(*Nocken speichern und Rest ignorieren*)
IF	fb_ton_end.Q AND
	(MEMCMP(ADR(gst_datensatz_copy.st_wkz.nockenschaltwerk_bestueckachse), ADR(gst_datensatz.st_wkz.nockenschaltwerk_bestueckachse), SIZEOF(gst_datensatz_copy.st_wkz.nockenschaltwerk_bestueckachse)) <> 0 ) THEN
	FOR j := 0 TO MAX_NOCKENGERUEST DO	(*nur die Nocken begin und end speichern*)
		IF	gst_datensatz_copy.st_wkz.nockenschaltwerk_bestueckachse.arr_nocken[j].r_cam_begin<>gst_datensatz.st_wkz.nockenschaltwerk_bestueckachse.arr_nocken[j].r_cam_begin OR
			gst_datensatz_copy.st_wkz.nockenschaltwerk_bestueckachse.arr_nocken[j].r_cam_end<>gst_datensatz.st_wkz.nockenschaltwerk_bestueckachse.arr_nocken[j].r_cam_end THEN
			i16_auftrag:=SCHREIBE_WKZ;
		END_IF
	END_FOR
	gst_datensatz_copy.st_wkz.nockenschaltwerk_bestueckachse:=gst_datensatz.st_wkz.nockenschaltwerk_bestueckachse;
END_IF

(*Wkz Daten speichern*)
IF	fb_ton_end.Q AND
	gi16_maschinenstatusinfo <> STATUS_MASCHINE_ARBEITET AND
	(MEMCMP(ADR(gst_datensatz_copy.st_wkz), ADR(gst_datensatz.st_wkz), SIZEOF(gst_datensatz_copy.st_wkz)) <> 0 ) THEN
	i16_auftrag:=SCHREIBE_WKZ;
END_IF

(*Band Daten speichern*)
IF	fb_ton_end.Q AND
	gi16_maschinenstatusinfo <> STATUS_MASCHINE_ARBEITET AND
	(MEMCMP(ADR(gst_datensatz_copy.st_band), ADR(gst_datensatz.st_band), SIZEOF(gst_datensatz_copy.st_band)) <> 0 ) THEN
	i16_auftrag:=SCHREIBE_BAND;
END_IF

(*Wt Daten speichern*)
IF	fb_ton_end.Q AND
	gi16_maschinenstatusinfo <> STATUS_MASCHINE_ARBEITET AND
	(MEMCMP(ADR(gst_datensatz_copy.st_wt), ADR(gst_datensatz.st_wt), SIZEOF(gst_datensatz_copy.st_wt)) <> 0 ) THEN
	i16_auftrag:=SCHREIBE_WT;
END_IF

(*Maschinen Daten speichern*)
IF	fb_ton_end.Q AND
	gi16_maschinenstatusinfo <> STATUS_MASCHINE_ARBEITET AND
	(MEMCMP(ADR(gst_datensatz_copy.st_md), ADR(gst_datensatz.st_md), SIZEOF(gst_datensatz_copy.st_md)) <> 0 ) THEN
	i16_auftrag:=SCHREIBE_MD;
	hm_md_speichern:=FALSE;
END_IF
END_ACTION
ACTION generiere_bestueckbild:
(* Step 1: erzeuge eine Liste mit allen unseren Pins *)
st_akt_bestueckprogramm.i32_anzahl := 0;

FOR i := 0 TO gst_bestueckbild.i32_anzahl_pins - 1 BY 1
DO
	IF (gst_bestueckbild.st_pins[i].typ = gst_datensatz.st_md.s_aktuelles_band) THEN
		st_akt_bestueckprogramm.lr_y[st_akt_bestueckprogramm.i32_anzahl] := gst_bestueckbild.st_pins[i].lr_y;
		st_akt_bestueckprogramm.lr_z[st_akt_bestueckprogramm.i32_anzahl] := gst_bestueckbild.st_pins[i].lr_z;
		st_akt_bestueckprogramm.i16_b[st_akt_bestueckprogramm.i32_anzahl] := 1;

		st_akt_bestueckprogramm.i32_anzahl  := st_akt_bestueckprogramm.i32_anzahl + 1;
	END_IF
END_FOR


(* Step 2: Sortieren: Bubblesort by Z *)
sort_akt();

(* Einragen in die globale Sruktur *)
gst_datensatz.st_bestueckprogramm := st_akt_bestueckprogramm;
gst_datensatz.st_md.s_aktueller_isk := gst_bestueckbild.s_isknummer;
END_ACTION
ACTION Hub_Faktor_ermitteln:
 (*ermitteln der maximal zu bestückenden Pins eines Bestückbildes=========================*)

FOR n := 0 TO 14 DO
	s_HelpBand[n]:='';
	i32_Anzahl[n]:=0;
END_FOR
i32_maxAnzahl := 0;

FOR n := 0 TO 14 DO
	FOR m := 0 TO gst_bestueckbild.i32_anzahl_pins - 1 DO
		IF	gst_bestueckbild.st_pins[m].typ <> s_HelpBand[0] AND
			gst_bestueckbild.st_pins[m].typ <> s_HelpBand[1] AND
			gst_bestueckbild.st_pins[m].typ <> s_HelpBand[2] AND
			gst_bestueckbild.st_pins[m].typ <> s_HelpBand[3] AND
			gst_bestueckbild.st_pins[m].typ <> s_HelpBand[4] AND
			gst_bestueckbild.st_pins[m].typ <> s_HelpBand[5] AND
			gst_bestueckbild.st_pins[m].typ <> s_HelpBand[6] AND
			gst_bestueckbild.st_pins[m].typ <> s_HelpBand[7] AND
			gst_bestueckbild.st_pins[m].typ <> s_HelpBand[8] AND
			gst_bestueckbild.st_pins[m].typ <> s_HelpBand[9] AND
			gst_bestueckbild.st_pins[m].typ <> s_HelpBand[10] AND
			gst_bestueckbild.st_pins[m].typ <> s_HelpBand[11] AND
			gst_bestueckbild.st_pins[m].typ <> s_HelpBand[12] AND
			gst_bestueckbild.st_pins[m].typ <> s_HelpBand[13] AND
			gst_bestueckbild.st_pins[m].typ <> s_HelpBand[14] THEN
			s_HelpBand[n]:=gst_bestueckbild.st_pins[m].typ;
		END_IF
	END_FOR
END_FOR

FOR n := 0 TO 14 DO
	FOR m := 0 TO gst_bestueckbild.i32_anzahl_pins - 1 DO
		IF gst_bestueckbild.st_pins[m].typ = s_HelpBand[n] AND s_HelpBand[n] <>'' THEN
			i32_Anzahl[n]:=i32_Anzahl[n]+1;
		END_IF
	END_FOR
	IF	i32_Anzahl[n]>i32_maxAnzahl THEN
		i32_maxAnzahl:=i32_Anzahl[n];
	END_IF
END_FOR

(* Faktor für die Hubzahl*)
lr_min_FaktorHub:=100/gst_datensatz.st_wkz.r_auto;

IF	i32_maxAnzahl > 0  THEN

	lr_FaktorHub:=(DINT_TO_LREAL(st_akt_bestueckprogramm.i32_anzahl) / DINT_TO_LREAL(i32_maxAnzahl)) * 1.2;
	IF	lr_FaktorHub > 1 THEN
		lr_FaktorHub:=1;
	END_IF
	IF	lr_FaktorHub < lr_min_FaktorHub THEN 	(*Bestückgeschwindigkeit nur um maximal 100Hub verringern*)
		lr_FaktorHub:=lr_min_FaktorHub;
	END_IF
ELSE
	lr_FaktorHub:=1;
END_IF
END_ACTION
ACTION Hub_Faktor_ermitteln_halbauto:
 (*ermitteln der maximal zu bestückenden Pins eines Bestückbildes=========================*)
n:=-1;
i32_maxAnzahl := 0;
FOR n := 0 TO 14 DO
	i32_Anzahl[n]:=gst_bestueckbild_halbauto.Wkz[n].i32_anzahl;
	IF	i32_Anzahl[n]>i32_maxAnzahl THEN
		i32_maxAnzahl:=i32_Anzahl[n];
	END_IF
END_FOR

(* Faktor für die Hubzahl*)
lr_min_FaktorHub:=100/gst_datensatz.st_wkz.r_auto;

IF	i32_maxAnzahl > 0  THEN

	lr_FaktorHub:=(DINT_TO_LREAL(gst_datensatz.st_bestueckprogramm.i32_anzahl) / DINT_TO_LREAL(i32_maxAnzahl)) * 1.35;
	IF	lr_FaktorHub > 1 THEN
		lr_FaktorHub:=1;
	END_IF
	IF	lr_FaktorHub < lr_min_FaktorHub THEN 	(*Bestückgeschwindigkeit nur um maximal 100Hub verringern*)
		lr_FaktorHub:=lr_min_FaktorHub;
	END_IF
ELSE
	lr_FaktorHub:=1;
END_IF
END_ACTION
ACTION path:
IF	s_Projekt_path <> '' THEN
	IF	FIND(s_md_path,':') = 0 THEN
		s_md_path 	:= CONCAT(s_Projekt_path,s_md_path);
	END_IF
	IF	FIND(s_tools_path,':') = 0 THEN
		s_tools_path 	:= CONCAT(s_Projekt_path,s_tools_path);
	END_IF
END_IF
END_ACTION
ACTION sort_akt:
FOR i := st_akt_bestueckprogramm.i32_anzahl -1 TO 1  BY -1
DO
	FOR k := 0 TO i -1 BY 1
	DO
		CASE gst_bestueckbild.enu_richtung OF

			(* Y Spalte Minus nach Plus: Bei gleichem Y: Z minus nach Plus *)
			YMinus_nach_YPlus_ZMinus_nach_ZPlus:
				IF F_Vergleich_LReal(st_akt_bestueckprogramm.lr_y[k+1] , st_akt_bestueckprogramm.lr_y[k]) THEN
					b_sort_swap := st_akt_bestueckprogramm.lr_z[k+1] < st_akt_bestueckprogramm.lr_z[k];
				ELSE
					b_sort_swap := st_akt_bestueckprogramm.lr_y[k+1] < st_akt_bestueckprogramm.lr_y[k];
				END_IF

			(* Y Spalte Minus nach Plus: Bei gleichem Y: Z Plus nach Minus *)
			YMinus_nach_YPlus_ZPlus_nach_ZMinus:
				IF F_Vergleich_LReal(st_akt_bestueckprogramm.lr_y[k+1] , st_akt_bestueckprogramm.lr_y[k]) THEN
					b_sort_swap := st_akt_bestueckprogramm.lr_z[k+1] > st_akt_bestueckprogramm.lr_z[k];
				ELSE
					b_sort_swap := st_akt_bestueckprogramm.lr_y[k+1]< st_akt_bestueckprogramm.lr_y[k];
				END_IF

			(* Y Spalte Plus nach Minus: Bei gleichem Y: Z Minus nach Plus *)
			YPlus_nach_YMinus_ZMinus_nach_ZPlus:
				IF F_Vergleich_LReal(st_akt_bestueckprogramm.lr_y[k+1] , st_akt_bestueckprogramm.lr_y[k]) THEN
					b_sort_swap := st_akt_bestueckprogramm.lr_z[k+1] < st_akt_bestueckprogramm.lr_z[k];
				ELSE
					b_sort_swap := st_akt_bestueckprogramm.lr_y[k+1] > st_akt_bestueckprogramm.lr_y[k];
				END_IF

			(* Y Spalte Plus nach Minus: Bei gleichem Y: Z Plus nach Minus *)
			YPlus_nach_YMinus_ZPlus_nach_ZMinus:
				IF F_Vergleich_LReal(st_akt_bestueckprogramm.lr_y[k+1] , st_akt_bestueckprogramm.lr_y[k]) THEN
					b_sort_swap := st_akt_bestueckprogramm.lr_z[k+1] > st_akt_bestueckprogramm.lr_z[k];
				ELSE
					b_sort_swap := st_akt_bestueckprogramm.lr_y[k+1] > st_akt_bestueckprogramm.lr_y[k];
				END_IF
		END_CASE

		IF b_sort_swap THEN
			(* Tauschen k + 1 <--> k *)
			swap_a := k; swap_b := k+1;	swap_in_akt();
		END_IF

	END_FOR
END_FOR
END_ACTION
ACTION subr_Wkz_Band_Wt_schreiben:
(* ======================================Schrittkette======================================== *)
fb_state_entry2(	i16_pos:= 1 );

CASE fb_state_entry2.i16_step OF
(*=======================================================*)
	0:

		fb_wkz_band_wt_schreiben.Start := FALSE;

		(*-----------------------Weiterschaltbedingungen----------------------------*)
		fb_state_entry2.i16_next_step := BEREIT;

(*=======================================================*)
	BEREIT:	(* Warte auf Änderung *)

		(*-----------------------Weiterschaltbedingungen----------------------------*)
		IF gst_datensatz.st_md.s_aktuelles_wkz <> s_name_alt_wkz OR
		    gst_datensatz.st_md.s_aktuelles_band <> s_name_alt_band OR
		    gst_datensatz.st_md.s_aktueller_wt <> s_name_alt_wt THEN
			s_name_alt_wkz := gst_datensatz.st_md.s_aktuelles_wkz;
			s_name_alt_band :=gst_datensatz.st_md.s_aktuelles_band;
			s_name_alt_wt := gst_datensatz.st_md.s_aktueller_wt;
			fb_state_entry2.i16_next_step := 200;
		END_IF

(*=======================================================*)
	200: (* Aktuelles WKZ in txt Datei schreiben *)
		IF fb_state_entry2.E THEN
			fb_wkz_band_wt_schreiben.ExportStr := gst_datensatz.st_md.s_aktuelles_wkz;
			fb_wkz_band_wt_schreiben.FileName := 'Aktuelles_Wkz.txt';
			fb_wkz_band_wt_schreiben.Start := TRUE;
		END_IF

		(*-----------------------Weiterschaltbedingungen----------------------------*)
		IF fb_wkz_band_wt_schreiben.Busy THEN
			fb_wkz_band_wt_schreiben.Start := FALSE;
			fb_state_entry2.i16_next_step := 210;
		END_IF

(*=======================================================*)
	210: (* warte auf fertig *)

		(*-----------------------Weiterschaltbedingungen----------------------------*)
		IF fb_wkz_band_wt_schreiben.Done THEN
			fb_state_entry2.i16_next_step := 300;
		END_IF

(*=======================================================*)
	300: (* Aktuelles WKZ in txt Datei schreiben *)
		IF fb_state_entry2.E THEN
			fb_wkz_band_wt_schreiben.ExportStr := gst_datensatz.st_md.s_aktuelles_band;
			fb_wkz_band_wt_schreiben.FileName := 'Aktuelles_Band.txt';
			fb_wkz_band_wt_schreiben.Start := TRUE;
		END_IF

		(*-----------------------Weiterschaltbedingungen----------------------------*)
		IF fb_wkz_band_wt_schreiben.Busy THEN
			fb_wkz_band_wt_schreiben.Start := FALSE;
			fb_state_entry2.i16_next_step := 310;
		END_IF

(*=======================================================*)
	310: (* warte auf fertig *)

		(*-----------------------Weiterschaltbedingungen----------------------------*)
		IF fb_wkz_band_wt_schreiben.Done THEN
			fb_state_entry2.i16_next_step := 400;
		END_IF

(*=======================================================*)
	400: (* Aktuellen Wt in txt Datei schreiben *)
		IF fb_state_entry2.E THEN
			fb_wkz_band_wt_schreiben.ExportStr := gst_datensatz.st_md.s_aktueller_wt;
			fb_wkz_band_wt_schreiben.FileName := 'Aktueller_Wt.txt';
			fb_wkz_band_wt_schreiben.Start := TRUE;
		END_IF

		(*-----------------------Weiterschaltbedingungen----------------------------*)
		IF fb_wkz_band_wt_schreiben.Busy THEN
			fb_wkz_band_wt_schreiben.Start := FALSE;
			fb_state_entry2.i16_next_step := 410;
		END_IF

(*=======================================================*)
	410: (* warte auf fertig *)

		(*-----------------------Weiterschaltbedingungen----------------------------*)
		IF fb_wkz_band_wt_schreiben.Done THEN
			fb_state_entry2.i16_next_step := BEREIT;
		END_IF

END_CASE

fb_state_entry2(i16_pos:= 2 );

fb_wkz_band_wt_schreiben(
	Start:= ,
	ExportStr:= ,
	FileName:= ,
	Path:= 'D:\BBgen\',
	Mode:= 2,
	Ready=> , 
	Busy=> , 
	Done=> ,
	Error=> );
END_ACTION
ACTION swap_in_akt:
lr_tmp := st_akt_bestueckprogramm.lr_y[swap_a];
st_akt_bestueckprogramm.lr_y[swap_a] := st_akt_bestueckprogramm.lr_y[swap_b];
st_akt_bestueckprogramm.lr_y[swap_b] := lr_tmp;

lr_tmp := st_akt_bestueckprogramm.lr_z[swap_a];
st_akt_bestueckprogramm.lr_z[swap_a] := st_akt_bestueckprogramm.lr_z[swap_b];
st_akt_bestueckprogramm.lr_z[swap_b] := lr_tmp;

i16_tmp := st_akt_bestueckprogramm.i16_b[swap_a];
st_akt_bestueckprogramm.i16_b[swap_a] := st_akt_bestueckprogramm.i16_b[swap_b];
st_akt_bestueckprogramm.i16_b[swap_b] := i16_tmp;
END_ACTION
ACTION wkz_gruppe_kompatibel:
(*Gruppe löschen wenn ein neues Werkzeug ausgewählt wird*)
IF	gst_datensatz_copy.st_md.s_aktuelles_wkz<>gst_datensatz.st_md.s_aktuelles_wkz THEN
	i:=-1;
	FOR i := 0 TO 4 DO
		gst_datensatz.st_md.st_wkz_gruppe[i].s_wkz := '';
		gst_datensatz.st_md.st_wkz_gruppe[i].i16_wkz_gruppe_kompatibel := 0;
		gst_datensatz.st_md.st_wkz_gruppe[i].s_Band := '';
		gst_datensatz.st_md.st_wkz_gruppe[i].i32_Wkz_nr := -1;
		gst_datensatz.st_md.st_wkz_gruppe[i].i32_Anzahl := -1;
	END_FOR
END_IF

(*Fehler*)
IF	state =0 THEN
	k:=-1;
	sm_Wkz_Gruppe_nicht_zugeordnet:=FALSE;
	sm_Wkz_nicht_kompatibel:=FALSE;
	FOR k := 0 TO 4 DO
		i:=-1;
		FOR i := 0 TO 4 DO
			IF	gst_datensatz.st_md.st_wkz_gruppe[k].s_wkz <> '' AND
				gst_datensatz.st_md.st_wkz_gruppe[i].s_wkz <> '' AND
				gst_datensatz.st_md.st_wkz_gruppe[k].i16_wkz_gruppe_kompatibel <>gst_datensatz.st_md.st_wkz_gruppe[i].i16_wkz_gruppe_kompatibel THEN
				sm_Wkz_nicht_kompatibel:=TRUE;
			END_IF
		END_FOR

		IF	gst_datensatz.st_md.st_wkz_gruppe[k].s_wkz <> '' AND
			gst_datensatz.st_md.st_wkz_gruppe[k].i16_wkz_gruppe_kompatibel = 0 THEN
			sm_Wkz_Gruppe_nicht_zugeordnet:=TRUE;
		END_IF

	END_FOR
END_IF

(*==========================================================================================*)
b_Wkz_Gruppe_gebildet:=
	NOT sm_Wkz_nicht_kompatibel AND
	gst_datensatz.st_md.st_wkz_gruppe[0].s_wkz <> '' AND
	gst_datensatz.st_md.st_wkz_gruppe[1].s_wkz <> '';

i16_anzahl_Wkz_Gruppen:=0;
k:=-1;
FOR k := 0 TO 4 DO
	IF	gst_datensatz.st_md.st_wkz_gruppe[k].s_wkz <> ''	THEN
		i16_anzahl_Wkz_Gruppen:=i16_anzahl_Wkz_Gruppen + 1;
	END_IF
END_FOR

(*==========================================================================================*)
CASE state OF
0:	(* Auslesen wenn ein neues Wkz ausgewählt wird*)
	fb_xml_srv_read.bExecute:= FALSE;
	k:=-1;
	FOR k := 0 TO 4 DO
		IF	state =0 AND
			st_wkz_gruppe_copy[k].s_wkz<>gst_datensatz.st_md.st_wkz_gruppe[k].s_wkz THEN

			IF	gst_datensatz.st_md.st_wkz_gruppe[k].s_wkz='' THEN
				st_wkz_gruppe_copy[k].s_wkz:=gst_datensatz.st_md.st_wkz_gruppe[k].s_wkz;
			ELSE
				i32_neues_Wkz:=k;
				state:=10;
			END_IF

			gst_datensatz.st_md.st_wkz_gruppe[k].i16_wkz_gruppe_kompatibel:=0;
			st_wkz_gruppe_copy[k].i16_wkz_gruppe_kompatibel:=0;
			gst_datensatz.st_md.st_wkz_gruppe[k].s_Band := '';
			gst_datensatz.st_md.st_wkz_gruppe[k].i32_Wkz_nr := -1;
			gst_datensatz.st_md.st_wkz_gruppe[k].i32_Anzahl := -1;

		END_IF
	END_FOR

10:	(*Start auslesen*)
	nErrId := 0;
	fb_xml_srv_read.sFilePath:= 'D:\BBgen\Wkz\';
	fb_xml_srv_read.sFilePath:= CONCAT(fb_xml_srv_read.sFilePath,gst_datensatz.st_md.st_wkz_gruppe[i32_neues_Wkz].s_wkz);
	fb_xml_srv_read.sFilePath:= CONCAT(fb_xml_srv_read.sFilePath,'.xml');
	fb_xml_srv_read.sXPath := '/root/gst_datensatz.st_wkz/I16_WKZ_GRUPPE_KOMPATIBEL';
	fb_xml_srv_read.sSymName:= '.gst_datensatz.st_md.st_wkz_gruppe[';
	fb_xml_srv_read.sSymName:= CONCAT(fb_xml_srv_read.sSymName,DINT_TO_STRING(i32_neues_Wkz));
	fb_xml_srv_read.sSymName:= CONCAT(fb_xml_srv_read.sSymName,'].i16_wkz_gruppe_kompatibel');
	fb_xml_srv_read.bExecute:= TRUE;

	IF fb_xml_srv_read.bBusy THEN
		fb_xml_srv_read.bExecute:= FALSE;
		state := 20;
	END_IF

20:	(* Lesevorgang erfolgreich? *)
	IF NOT fb_xml_srv_read.bBusy THEN
		IF NOT fb_xml_srv_read.bError THEN
			state := 0;
			st_wkz_gruppe_copy[i32_neues_Wkz].s_wkz:=gst_datensatz.st_md.st_wkz_gruppe[i32_neues_Wkz].s_wkz;
			st_wkz_gruppe_copy[i32_neues_Wkz].i16_wkz_gruppe_kompatibel:=gst_datensatz.st_md.st_wkz_gruppe[i32_neues_Wkz].i16_wkz_gruppe_kompatibel;
		ELSE	(* Fehler *)
			nErrId := fb_xml_srv_read.nErrId;
			state := FEHLER;
		END_IF
	END_IF

FEHLER:
	state := 0;
	st_wkz_gruppe_copy[i32_neues_Wkz].s_wkz:=gst_datensatz.st_md.st_wkz_gruppe[i32_neues_Wkz].s_wkz;
END_CASE
END_ACTION

(* POU EPT Lib/Funktionsbausteine/ST_StateEntry, ST *)
FUNCTION_BLOCK ST_StateEntry
VAR
	arr_last_step_history	: ARRAY[0..31] OF STRING(110);
	i 					: INT := 0;
	last_pos 				: INT := 0;
	interner_step			: INT := 0;
	s_stepTime 			: STRING;
END_VAR
VAR_OUTPUT
	i16_last_step 			: enum_step_nr := INIT_OBJ;	(* Der Schritt vor diesem Schritt *)
	i16_step 				: enum_step_nr := INIT_OBJ;	(* Diese variable soll vom "case step of" verwendet werden *)
	E					: BOOL;					(* Aktiv bei betreten des Steps *)
	X					: BOOL;					(* Aktiv beim verlassen des Steps *)
	b_error 				: BOOL := FALSE;			(* Ablauf Pos 1,2,1,2,1,2,... nicht richtig *)
	fb_ton_Step			: TON;
END_VAR
VAR_INPUT
	i16_next_step 		: enum_step_nr := INIT_OBJ;	(* Nächster schritt *)
	i16_pos 				: INT;					(* Pos = 1: Aufruf vor dem Case step of ---  Pos = 2: Aufruf nach dem Case step of*)
	s_debugtext			: STRING(100);
END_VAR
VAR CONSTANT
	t_MaxStepTime		: TIME := T#60S;
END_VAR
(*stepTime ermitteln*)
fb_ton_Step(IN:= , PT:=t_MaxStepTime , Q=>  , ET=> );
IF	i16_step = i16_next_step THEN
	fb_ton_Step.IN:=TRUE;
END_IF

IF NOT b_error THEN
	CASE interner_step OF
		0:
			(* Mitten im Schritt drin *)
			X := FALSE;
			E := FALSE;


			(* Schritt wird verlassen *)
			IF i16_step <> i16_next_step AND i16_pos = 1 THEN
				subrDebugtext();
				interner_step := 10;
				X := TRUE;
				E := FALSE;
				fb_ton_Step.IN:=FALSE;
			END_IF

		10:
			(* Eintritt in neuen Schritt *)
			IF i16_pos = 1 THEN
				X := FALSE;
				E := TRUE;

				(* Schalte Schritt weiter *)
				i16_last_step := i16_step;
				i16_step := i16_next_step;
				(* Baue Statehistory *)

				IF  E THEN
					FOR i:= 31 TO 1 BY -1 DO
						arr_last_step_history[i] := arr_last_step_history[i-1];
					END_FOR
					arr_last_step_history[0] := '';
					s_stepTime:='';
					s_debugtext:='';
				END_IF

				interner_step := 0;

			END_IF
	END_CASE
END_IF

IF 	(fb_ton_Step.ET >= T#200ms AND arr_last_step_history[0] = '') OR	(* Am Anfang Debugtext schreiben, damit etwas drin steht *)
	(fb_ton_Step.Q AND s_stepTime <> '>1m') THEN	(* Debugtext schreiben, wenn t_MaxStepTime erreicht wird *)
	subrDebugtext();
END_IF

(* Prüfe Baustein *)
IF 	i16_pos = last_pos THEN
	b_error := TRUE;
END_IF

last_pos := i16_pos;
END_FUNCTION_BLOCK
ACTION subrDebugtext:
s_stepTime:=ET_TO_STRING(fb_ton_Step.ET);
IF 	fb_ton_Step.ET >= t_MaxStepTime THEN
	s_stepTime:=CONCAT('>',s_StepTime);
END_IF

(* history zusammenbauen aus StepNr, StepTime und debugtext*)
CASE i16_step OF
	INIT_OBJ :			arr_last_step_history[0]:='INIT_OBJ';
	INIT :				arr_last_step_history[0]:='INIT';
	BEREIT :				arr_last_step_history[0]:='BEREIT';
	FEHLER :			arr_last_step_history[0]:='FEHLER';
	STOP :				arr_last_step_history[0]:='STOP';
	STILLSTAND :		arr_last_step_history[0]:='STILLSTAND';
	HALT :				arr_last_step_history[0]:='HALT';
	HANDRAD :			arr_last_step_history[0]:='HANDRAD';
	MOTORBREMSE_AUF :	arr_last_step_history[0]:='MOTORBREMSE_AUF';
	MOTORBREMSE_ZU :	arr_last_step_history[0]:='MOTORBREMSE_ZU';
	LUEFTEN :			arr_last_step_history[0]:='LUEFTEN';
	REGELN :			arr_last_step_history[0]:='REGELN';
	INBETRIEBNAHME :		arr_last_step_history[0]:='INBETRIEBNAHME';
	(* Zylinder *)
	ZYL_INIT :			arr_last_step_history[0]:='ZYL_INIT';
	GESTOPPT :			arr_last_step_history[0]:='GESTOPPT';
	EINGEFAHREN :		arr_last_step_history[0]:='EINGEFAHREN';
	BEWEGUNG_AUSFAHREN :		arr_last_step_history[0]:='BEWEGUNG_AUSFAHREN';
	AUSGEFAHREN :		arr_last_step_history[0]:='AUSGEFAHREN';
	BEWEGUNG_EINFAHREN :		arr_last_step_history[0]:='BEWEGUNG_EINFAHREN';
	MITTEGEFAHREN :		arr_last_step_history[0]:='MITTEGEFAHREN';
	BEWEGUNG_MITTE  :	arr_last_step_history[0]:='BEWEGUNG_MITTE';
	LUFTLOS :			arr_last_step_history[0]:='LUFTLOS';
	ZYL_FEHLER :		arr_last_step_history[0]:='ZYL_FEHLER';
	DIREKT_EINFAHREN :	arr_last_step_history[0]:='DIREKT_EINFAHREN';
	DIREKT_AUSFAHREN :	arr_last_step_history[0]:='DIREKT_AUSFAHREN';
ELSE
	arr_last_step_history[0] := INT_TO_STRING(i16_step);
END_CASE

IF 	s_stepTime ='0ms' OR s_stepTime =''THEN
	s_stepTime:='3ms';		(*damit nicht 0 drin steht*)
END_IF
arr_last_step_history[0] := CONCAT(arr_last_step_history[0],':  ');
arr_last_step_history[0] := CONCAT(arr_last_step_history[0],s_stepTime);
arr_last_step_history[0] := CONCAT(arr_last_step_history[0],': ');
arr_last_step_history[0] := CONCAT(arr_last_step_history[0],s_debugtext);
END_ACTION

(* POU EPT Lib/Funktionen/ET_TO_STRING, ST *)
FUNCTION ET_TO_STRING :STRING
VAR_INPUT
	et		:TIME;
END_VAR

VAR
	i16_LEN	:INT;
END_VAR
ET_TO_STRING:=TIME_TO_STRING(et);
ET_TO_STRING:=DELETE(ET_TO_STRING,2,1);

IF 	et> t#60s THEN
	ET_TO_STRING:=LEFT(ET_TO_STRING,FIND(ET_TO_STRING,'s'));
END_IF
END_FUNCTION

(* POU Gemeinsamkeiten17xx/BBGen/ST_BBGenXMLFile, ST *)
FUNCTION_BLOCK ST_BBGenXMLFile
VAR_INPUT
	bQuit								: BOOL;
	(* ISK *)
	start_lesen_isk						: BOOL;
	start_schreiben_isk					: BOOL;

	(* Wkz *)
	start_lesen_wkz						: BOOL;
	start_schreiben_wkz					: BOOL;

	(* Bestueckbild wird nur gelesen *)
	start_lesen_bestueckbild				: BOOL;
	start_schreiben_bestueckbild			: BOOL;

	(* Bestueckbild Halbautomatik wird nur gelesen *)
	start_lesen_bestueckbild_halbauto				: BOOL;
	start_schreiben_bestueckbild_halbauto			: BOOL;

	(* Maschinendaten *)
	start_lesen_md						: BOOL;
	start_schreiben_md					: BOOL;
	start_schreiben_md_backup			: BOOL;

	(* Banddaten *)
	start_lesen_band						: BOOL;
	start_schreiben_band					: BOOL;

	(* Wt-Daten *)
	start_lesen_wt						: BOOL;
	start_schreiben_wt						: BOOL;

	(* Wo liegen die Dateien *)
	s_path								: STRING(255);

	(* Welche Dateien? *)
	s_bestueckbild						: STRING(50);
	s_wkz								: STRING(50);
	s_isk								: STRING(50);
	s_md								: STRING(50);
	s_md_backup						: STRING(50);
	s_band								: STRING(50);
	s_wt									: STRING(50);
END_VAR
VAR_OUTPUT
	fertig_lesen							: BOOL;
	fertig_schreiben						: BOOL;

	bError								: BOOL;
	nErrId								: UDINT;
END_VAR
VAR
	fb_state_entry							: ST_StateEntry;
	fb_ton_quitt							: TON;
	fb_xml_srv_write						: FB_XmlSrvWriteByName;
	fb_xml_srv_read						: FB_XmlSrvReadByName;
	s_file								: STRING(255);

END_VAR
fb_ton_quitt(IN:= , PT:= t#50ms, Q=> , ET=> );

(* ======================================Schrittkette======================================== *)
fb_state_entry(
	i16_next_step:= ,
	i16_pos:= 1,
	s_debugtext:= ,
	E=> ,
	X=> ,
	i16_step=> ,
	i16_last_step=> );


CASE fb_state_entry.i16_step OF
(*=======================================================*)
	0:
		bError := FALSE;
		nErrId := 0;

		fertig_lesen := FALSE;
		fertig_schreiben := FALSE;

		fb_state_entry.i16_next_step := 10;

(*=======================================================*)
	10:	(* Auslesen der Daten aus den XML-Files *)
		(* Daten lesen *)
		IF start_lesen_isk THEN
			s_file := CONCAT(s_path, s_isk);
			s_file := CONCAT(s_file,'.xml');
			fb_xml_srv_read.sSymName := '.gst_datensatz.st_isk';
			fb_xml_srv_read.sXPath := '/root/gst_datensatz.st_isk';
			fb_state_entry.i16_next_step := 100;
		ELSIF start_lesen_bestueckbild THEN
			s_file := CONCAT(s_path, s_bestueckbild);
			s_file := CONCAT(s_file,'.xml');
			fb_xml_srv_read.sSymName := '.gst_bestueckbild';
			fb_xml_srv_read.sXPath := '/root/gst_bestueckbild';
			fb_state_entry.i16_next_step := 100;

		ELSIF start_lesen_bestueckbild_halbauto THEN
			s_file := CONCAT(s_path, s_bestueckbild);
			s_file := CONCAT(s_file,'.xml');
			fb_xml_srv_read.sSymName := '.gst_bestueckbild_halbauto';
			fb_xml_srv_read.sXPath := '/root/gst_bestueckbild_halbauto';
			fb_state_entry.i16_next_step := 100;

		ELSIF start_lesen_wkz THEN
			s_file := CONCAT(s_path, s_wkz);
			s_file := CONCAT(s_file,'.xml');
			fb_xml_srv_read.sSymName := '.gst_datensatz.st_wkz';
			fb_xml_srv_read.sXPath := '/root/gst_datensatz.st_wkz';
			fb_state_entry.i16_next_step := 100;
		ELSIF start_lesen_md THEN
			s_file := CONCAT(s_path, s_md);
			s_file := CONCAT(s_file,'.xml');
			fb_xml_srv_read.sSymName := '.gst_datensatz.st_md';
			fb_xml_srv_read.sXPath := '/root/gst_datensatz.st_md';
			fb_state_entry.i16_next_step := 100;
		ELSIF start_lesen_band THEN
			s_file := CONCAT(s_path, s_band);
			s_file := CONCAT(s_file,'.xml');
			fb_xml_srv_read.sSymName := '.gst_datensatz.st_band';
			fb_xml_srv_read.sXPath := '/root/gst_datensatz.st_band';
			fb_state_entry.i16_next_step := 100;
		ELSIF start_lesen_wt THEN
			s_file := CONCAT(s_path, s_wt);
			s_file := CONCAT(s_file,'.xml');
			fb_xml_srv_read.sSymName := '.gst_datensatz.st_wt';
			fb_xml_srv_read.sXPath := '/root/gst_datensatz.st_wt';
			fb_state_entry.i16_next_step := 100;
		END_IF

		(* Daten schreiben *)
		IF start_schreiben_isk THEN
			s_file := CONCAT(s_path, s_isk);
			s_file := CONCAT(s_file,'.xml');
			fb_xml_srv_write.sSymName := '.gst_datensatz.st_isk';
			fb_xml_srv_write.sXPath := '/root/gst_datensatz.st_isk';
			fb_state_entry.i16_next_step := 200;
		ELSIF start_schreiben_bestueckbild THEN
			s_file := CONCAT(s_path, s_bestueckbild);
			s_file := CONCAT(s_file,'.xml');
			fb_xml_srv_write.sSymName := '.gst_bestueckbild';
			fb_xml_srv_write.sXPath := '/root/gst_bestueckbild';
			fb_state_entry.i16_next_step := 200;
		ELSIF start_schreiben_bestueckbild_halbauto THEN
			s_file := CONCAT(s_path, s_bestueckbild);
			s_file := CONCAT(s_file,'.xml');
			fb_xml_srv_write.sSymName := '.gst_bestueckbild_halbauto';
			fb_xml_srv_write.sXPath := '/root/gst_bestueckbild_halbauto';
			fb_state_entry.i16_next_step := 200;
		ELSIF start_schreiben_wkz THEN
			s_file := CONCAT(s_path, s_wkz);
			s_file := CONCAT(s_file,'.xml');
			fb_xml_srv_write.sSymName := '.gst_datensatz.st_wkz';
			fb_xml_srv_write.sXPath := '/root/gst_datensatz.st_wkz';
			fb_state_entry.i16_next_step := 200;
		ELSIF start_schreiben_md_backup THEN
			s_file := CONCAT(s_path, s_md_backup);
			s_file := CONCAT(s_file,'.xml');
			fb_xml_srv_write.sSymName := '.gst_datensatz.st_md';
			fb_xml_srv_write.sXPath := '/root/gst_datensatz.st_md';
			fb_state_entry.i16_next_step := 200;
		ELSIF start_schreiben_md THEN
			s_file := CONCAT(s_path, s_md);
			s_file := CONCAT(s_file,'.xml');
			fb_xml_srv_write.sSymName := '.gst_datensatz.st_md';
			fb_xml_srv_write.sXPath := '/root/gst_datensatz.st_md';
			fb_state_entry.i16_next_step := 200;
		ELSIF start_schreiben_band THEN
			s_file := CONCAT(s_path, s_band);
			s_file := CONCAT(s_file,'.xml');
			fb_xml_srv_write.sSymName := '.gst_datensatz.st_band';
			fb_xml_srv_write.sXPath := '/root/gst_datensatz.st_band';
			fb_state_entry.i16_next_step := 200;
		ELSIF start_schreiben_wt THEN
			s_file := CONCAT(s_path, s_wt);
			s_file := CONCAT(s_file,'.xml');
			fb_xml_srv_write.sSymName := '.gst_datensatz.st_wt';
			fb_xml_srv_write.sXPath := '/root/gst_datensatz.st_wt';
			fb_state_entry.i16_next_step := 200;
		END_IF

(*=======================================================*)
	100:	(* Starte Daten lesen *)
		IF fb_state_entry.E THEN
			fb_xml_srv_read.bExecute := TRUE;
			fb_xml_srv_read.sFilePath := s_file;
		END_IF

		IF fb_xml_srv_read.bBusy THEN
			fb_xml_srv_read.bExecute := FALSE;
			fb_state_entry.i16_next_step := 110;
		END_IF

(*=======================================================*)
	110:	(* Lesevorgang *)
		IF NOT fb_xml_srv_read.bBusy  THEN
			IF NOT fb_xml_srv_read.bError THEN
				fb_state_entry.i16_next_step := 120;
			ELSE	(* Fehler *)
				nErrId := fb_xml_srv_read.nErrId;
				fb_state_entry.i16_next_step := 1000;
			END_IF
		END_IF

(*=======================================================*)
	120:	(* Lesevorgang beendet *)
		IF fb_state_entry.E THEN
			fertig_lesen := TRUE;
		END_IF

		IF 	NOT start_lesen_band AND
			NOT start_lesen_bestueckbild AND
			NOT start_lesen_isk AND
			NOT start_lesen_md AND
			NOT start_lesen_wkz AND
			NOT start_lesen_wt AND
			NOT fb_state_entry.E
			THEN
				fb_state_entry.i16_next_step := 0;
		END_IF

		IF fb_state_entry.X THEN
			fertig_lesen := TRUE;
		END_IF

(*=======================================================*)
	200:	(* Starte Daten schreiben *)
		IF fb_state_entry.E THEN
			fb_xml_srv_write.bExecute := TRUE;
			fb_xml_srv_write.sFilePath := s_file;
		END_IF

		IF fb_xml_srv_write.bBusy THEN
			fb_xml_srv_write.bExecute := FALSE;
			fb_state_entry.i16_next_step := 210;
		END_IF

(*=======================================================*)
	210:	(* Schreibvorgang *)
		IF NOT fb_xml_srv_write.bBusy  THEN
			IF NOT fb_xml_srv_write.bError THEN
				fb_state_entry.i16_next_step := 220;
			ELSE	(* Fehler *)
				nErrId := fb_xml_srv_write.nErrId;
				fb_state_entry.i16_next_step := 1000;
			END_IF
		END_IF

(*=======================================================*)
	220:	(* Schreibvorgang beendet *)
		IF fb_state_entry.E THEN
			fertig_schreiben := TRUE;
		END_IF

		IF 	NOT start_schreiben_band AND
			NOT start_schreiben_bestueckbild AND
			NOT start_schreiben_isk AND
			NOT start_schreiben_md AND
			NOT start_schreiben_md_backup AND
			NOT start_schreiben_wkz AND
			NOT start_schreiben_wt AND
			NOT fb_state_entry.E
			THEN
				fb_state_entry.i16_next_step := 0;
		END_IF

		IF fb_state_entry.X THEN
			fertig_schreiben := TRUE;
		END_IF

(*=======================================================*)
	1000: (* Fehler *)
		IF fb_state_entry.E THEN
			bError := TRUE;
			fb_ton_quitt.IN := FALSE;
		END_IF

		(*-----------------------Weiterschaltbedingungen----------------------------*)
		IF bQuit AND NOT fb_state_entry.E THEN
			bError := FALSE;
			fb_ton_quitt.IN := TRUE;
		END_IF

		IF fb_ton_quitt.Q THEN
			fb_ton_quitt.IN := FALSE;
			fb_state_entry.i16_next_step := 0;
		END_IF
END_CASE


fb_state_entry(
	i16_next_step:= ,
	i16_pos:= 2,
	s_debugtext:= ,
	E=> ,
	X=> ,
	i16_step=> ,
	i16_last_step=> );

(* XML *)
fb_xml_srv_read(
	sNetId:= '',
	ePath:= PATH_GENERIC,
	nMode:= XMLSRV_SKIPMISSING,
	sSymName:= ,
	sFilePath:= ,
	sXPath:= ,
	bExecute:= ,
	tTimeout:= t#10s,
	bBusy=> ,
	bError=> ,
	nErrId=> );

fb_xml_srv_write(
	sNetId:= '',
	ePath:= PATH_GENERIC,
	nMode:= XMLSRV_ADDMISSING,
	sSymName:=  ,
	sFilePath:= ,
	sXPath:= ,
	bExecute:= ,
	tTimeout:= t#10s,
	bBusy=> ,
	bError=> ,
	nErrId=> );
END_FUNCTION_BLOCK

(* POU Gemeinsamkeiten17xx/BBGen/ST_BBGenWriteFile, ST *)
FUNCTION_BLOCK ST_BBGenWriteFile
VAR_INPUT
	bStart		: BOOL;
END_VAR
VAR_OUTPUT
	bFertig	: BOOL;
	bError	: BOOL;
END_VAR
VAR
	fb_state_entry						: ST_StateEntry;
	fb_r_trig_start						: R_TRIG;
	fb_ton_quitt						: TON;
	fb_openfile						: FILEOPEN;
	fb_writefile						: FILEWRITE;
	fb_closefile						: FILECLOSE;

	s_file							: STRING(255);

	nErrId							: DINT;

	tmp								: DINT;
	lo								: DINT;
	ll								: DINT;
	s_line							: STRING(255);
	s_out							: STRING(10000);
	y								: STRING;
	z								: STRING;
	b								: STRING;
	tab								: STRING;
	lineend							: STRING;
END_VAR
fb_ton_quitt(IN:= , PT:= t#50ms, Q=> , ET=> );
fb_r_trig_start(CLK:= bStart, Q=> );
(* ======================================Schrittkette======================================== *)
fb_state_entry(
	i16_next_step:= ,
	i16_pos:= 1,
	s_debugtext:= ,
	E=> ,
	X=> ,
	i16_step=> ,
	i16_last_step=> );


CASE fb_state_entry.i16_step OF
(*=======================================================*)
	0:
		nErrId := 0;

		bFertig := FALSE;
		bError := FALSE;

		s_file := 'D:\BBGen\bbgen.txt';
		fb_state_entry.i16_next_step := 10;
(*=======================================================*)
	10:
		IF fb_r_trig_start.Q THEN
			fb_state_entry.i16_next_step := 100;
		END_IF
(*=======================================================*)
	100:
		(* Öffne Datei *)
		IF fb_state_entry.E THEN
			fb_openfile.OPEN := TRUE;
		END_IF

		IF fb_openfile.ERR THEN
			fb_state_entry.i16_next_step := FEHLER;
			nErrId := fb_openfile.ERRID;
		END_IF

		IF NOT fb_state_entry.E AND NOT fb_openfile.BUSY AND NOT fb_openfile.ERR THEN
			fb_state_entry.i16_next_step := 110;
		END_IF

		IF fb_state_entry.X THEN
			fb_openfile.OPEN := FALSE;
		END_IF
(*=======================================================*)
	110:
		(* Datei ist offen. Schreibe Einträge*)
		IF fb_state_entry.E THEN
			(* Baue Ausgabestring *)
			s_out := '';
			tab := '$T';
			lineend := '$R$N';
			lo := 0;
			ll := 0;
			(* Erste Zeile: Offset und Breite/Höhe*)
			y := LREAL_TO_FMTSTR(gst_datensatz.st_isk.lr_pos_y_0,2,TRUE);	s_line := CONCAT(y,tab);
			z := LREAL_TO_FMTSTR(gst_datensatz.st_isk.lr_pos_z_0,2,TRUE);	s_line := CONCAT(s_line,z);	s_line := CONCAT(s_line,tab);

			y := LREAL_TO_FMTSTR(gst_datensatz.st_isk.lr_breite,2,TRUE);		s_line := CONCAT(s_line,y);	s_line := CONCAT(s_line,tab);
			z := LREAL_TO_FMTSTR(gst_datensatz.st_isk.lr_hoehe,2,TRUE);		s_line := CONCAT(s_line,z);	s_line := CONCAT(s_line,lineend);
			s_out := s_line; lo := LEN(s_out);

			FOR tmp := 0 TO gst_datensatz.st_bestueckprogramm.i32_anzahl-1 BY 1
			DO
				y := LREAL_TO_FMTSTR (gst_datensatz.st_bestueckprogramm.lr_y[tmp],2,TRUE);
				z := LREAL_TO_FMTSTR(gst_datensatz.st_bestueckprogramm.lr_z[tmp],2,TRUE);
				b := INT_TO_STRING(gst_datensatz.st_bestueckprogramm.i16_b[tmp]);
				s_line := y;						ll := LEN(y);
				s_line := CONCAT(s_line, tab);		ll := ll + LEN(tab);
				s_line := CONCAT(s_line, z);			ll := ll + LEN(z);
				s_line := CONCAT(s_line, tab);		ll := ll + LEN(tab);
				s_line := CONCAT(s_line, b);			ll := ll + LEN(b);
				s_line := CONCAT(s_line, lineend);	ll := ll + LEN(lineend);

				(* Da concat und co nur Strings bis 255 Zeichen kann, müssen wir hier memcpy nutzen *)
				MEMCPY(ADR(s_out)+lo,ADR(s_line), ll);
				lo := lo + ll;
			END_FOR
			fb_writefile.BUFADDR := ADR(s_out);
			fb_writefile.COUNT := lo;
			fb_writefile.WRITE := TRUE;
		END_IF

		IF NOT fb_state_entry.E AND fb_writefile.ERR  THEN
			fb_state_entry.i16_next_step := FEHLER;
			nErrId := fb_writefile.ERRID;
		END_IF

		IF NOT fb_state_entry.E AND NOT fb_writefile.BUSY AND NOT fb_writefile.ERR THEN
			(* Erfolgreich geschrieben *)
			fb_state_entry.i16_next_step := 200;
		END_IF

		IF fb_state_entry.X THEN
			fb_writefile.WRITE := FALSE;
		END_IF

(*=======================================================*)
	200:
		(* Schliesse Datei *)
		IF fb_state_entry.E THEN
			fb_closefile.CLOSE := TRUE;
		END_IF

		IF fb_closefile.ERR THEN
			fb_state_entry.i16_next_step := FEHLER;
			nErrId := fb_closefile.ERRID;
		END_IF

		IF NOT fb_state_entry.E AND NOT fb_closefile.BUSY AND NOT fb_closefile.ERR THEN
			fb_state_entry.i16_next_step := 210;
		END_IF

		IF fb_state_entry.X THEN
			fb_closefile.CLOSE := FALSE;
		END_IF

(*=======================================================*)
	210:
		IF fb_state_entry.E THEN
			bFertig := TRUE;
		END_IF

		IF NOT bStart AND NOT fb_state_entry.E THEN
			fb_state_entry.i16_next_step := 10;
		END_IF

		IF fb_state_entry.X THEN
			bFertig := FALSE;
		END_IF

(*=======================================================*)
	1000: (* Fehler *)
		IF fb_state_entry.E THEN
			bError := TRUE;
			fb_ton_quitt.IN := FALSE;
		END_IF

		(*-----------------------Weiterschaltbedingungen----------------------------*)
		IF NOT fb_state_entry.E THEN
			bError := FALSE;
			fb_ton_quitt.IN := TRUE;
		END_IF

		IF fb_ton_quitt.Q THEN
			fb_ton_quitt.IN := FALSE;
			fb_state_entry.i16_next_step := 0;
		END_IF
END_CASE

fb_state_entry(
	i16_next_step:= ,
	i16_pos:= 2,
	s_debugtext:= ,
	E=> , 
	X=> ,
	i16_step=> ,
	i16_last_step=> );

(* FILE *)
fb_openfile(
	NETID:= ,
	FPATHNAME:= s_file,
	OPENMODE:= FILE_OPENWRITE, (* Wir wollen eine bestehenede Datei im Falle überschreiben *)
	OPEN:= ,
	TMOUT:= t#2s,
	BUSY=> , 
	ERR=> , 
	ERRID=> , 
	HFILE=> );

fb_writefile(
	NETID:= ,
	HFILE:= fb_openfile.HFILE,
	BUFADDR:= , 
	COUNT:= ,
	WRITE:= ,
	TMOUT:= t#2s,
	BUSY=> ,
	ERR=> ,
	ERRID=> ,
	COUNT_W=> );

fb_closefile(
	NETID:= , 
	HFILE:= fb_openfile.HFILE,
	CLOSE:= , 
	TMOUT:= t#2s,
	BUSY=> ,
	ERR=> , 
	ERRID=> );
END_FUNCTION_BLOCK

(* POU EPT Lib/Funktionsbausteine/ST_Export_String, ST *)
FUNCTION_BLOCK ST_Export_String
VAR_INPUT
	Start				:BOOL;
	ExportStr			:STRING(255);
	FileName			:STRING;
	Path				:STRING;
	Mode				:DWORD;
END_VAR
VAR
	fb_state_entry		:ST_StateEntry;
	fb_file_open			:FB_FileOpen;
	fb_file_puts			:FB_FilePuts;
	fb_file_close			:FB_FileClose;
	nErrId					:UDINT;
	ErrorMsg			:STRING(255);
	hFile				:UINT;
END_VAR
VAR_OUTPUT
	Ready				:BOOL;
	Busy				:BOOL;
	Done				:BOOL;
	Error				:BOOL;
END_VAR
fb_state_entry(i16_pos:= 1);

CASE fb_state_entry.i16_step OF

(*=======================================================*)
	0:	(*Objekt initialisieren*)

		(*-----------------------Weiterschaltbedingungen----------------------------*)
		fb_state_entry.i16_next_step:=INIT;

(*=======================================================*)
	10:	(*initialisieren*)

		(*-----------------------Weiterschaltbedingungen----------------------------*)
		fb_state_entry.i16_next_step:=BEREIT;

(*=======================================================*)
	BEREIT:(*Start*)

		(*-----------------------Weiterschaltbedingungen----------------------------*)
		IF Start THEN
			Start:=FALSE;
			Busy:=TRUE;
			Error:=FALSE;
			Done:=FALSE;
			nErrId:=0;
			ErrorMsg:='';
			fb_state_entry.i16_next_step:=105;
		END_IF

(*=======================================================*)
	105: (*Datei erstellen*)
		IF fb_state_entry.E THEN
			fb_file_open.sPathName:=CONCAT (Path, FileName);
			fb_file_open.bExecute:=TRUE;
		END_IF

		(*-----------------------Weiterschaltbedingungen----------------------------*)
		IF  fb_file_open.bBusy THEN
			fb_state_entry.i16_next_step:=110;
		END_IF

(*=======================================================*)
	110: (*Datei erstellen*)

		(*-----------------------Weiterschaltbedingungen----------------------------*)
		IF 	NOT fb_file_open.bBusy THEN
			fb_file_open.bExecute:=FALSE;
			IF 	fb_file_open.bError THEN
				nErrId:=fb_file_open.nErrId;
				fb_state_entry.i16_next_step:=FEHLER;
				ErrorMsg:='Fehler beim Öffnen der Datei';
			ELSE
				fb_state_entry.i16_next_step:=120;
			END_IF
		END_IF

(*=======================================================*)
	120: (*String in Datei eintragen*)
		IF fb_state_entry.E THEN
			fb_file_puts.sLine:=ExportStr;
			fb_file_puts.bExecute:=TRUE;
		END_IF

		(*-----------------------Weiterschaltbedingungen----------------------------*)
		IF  fb_file_puts.bBusy THEN
			fb_state_entry.i16_next_step:=130;
		END_IF

(*=======================================================*)
	130: (*String in Datei eintragen*)

		(*-----------------------Weiterschaltbedingungen----------------------------*)
		IF 	NOT fb_file_puts.bBusy THEN
			fb_file_puts.bExecute:=FALSE;
			IF 	fb_file_puts.bError THEN
				nErrId:=fb_file_puts.nErrId;
				fb_state_entry.i16_next_step:=FEHLER;
			ELSE
				fb_state_entry.i16_next_step:=140;
			END_IF
		END_IF
	
(*=======================================================*)
	140:(*Datei schließen*)
		IF fb_state_entry.E THEN
		fb_file_close.bExecute:=TRUE;
		END_IF

		(*-----------------------Weiterschaltbedingungen----------------------------*)
		IF 	fb_file_close.bBusy THEN
			fb_state_entry.i16_next_step:=150;
		END_IF
	
(*=======================================================*)
	150:(*Datei schließen*)

		(*-----------------------Weiterschaltbedingungen----------------------------*)
		IF NOT fb_file_close.bBusy THEN
			fb_file_close.bExecute:=FALSE;
			IF 	fb_file_close.bError THEN
				nErrId:=fb_file_close.nErrId;
				fb_state_entry.i16_next_step:=FEHLER;
				ErrorMsg:='Fehler beim Schließen der Datei';
			ELSE
				Busy:=FALSE;
				Done:=TRUE;
				fb_state_entry.i16_next_step:=BEREIT;
			END_IF
		END_IF

(*=======================================================*)
	FEHLER:	(*bei Fehler einfach weiter*)

		Busy:=FALSE;
		Error:=TRUE;
		fb_state_entry.i16_next_step := INIT;

END_CASE

fb_state_entry(i16_pos:= 2);


fb_file_open(
	sNetId:='',
	sPathName:= ,
	nMode:=Mode,
	ePath:=PATH_GENERIC,
	bExecute:= ,
	tTimeout:=T#1s,
	hFile=> hFile);

fb_file_puts(
	sNetId:='',
	hFile:=hFile,
	sLine:= ,
	bExecute:= ,
	tTimeout:=t#1s);

fb_file_close(
	sNetId:='',
	hFile:=hFile,
	bExecute:= ,
	tTimeout:=t#1s);
END_FUNCTION_BLOCK

(* POU Gemeinsamkeiten17xx/Safety/ST_Safetyprogramm, ST *)
PROGRAM ST_Safetyprogramm
VAR_INPUT
	st_config							: struct_config;
	st_ctrl_in							: struct_ctrl_in;
END_VAR
VAR_IN_OUT
	st_visu							: struct_visu;
END_VAR
VAR_OUTPUT
	st_ctrl_out						: struct_ctrl_out;
END_VAR
VAR
	ack_step							: ST_StateEntry;
	fb_ton_wz						: TON;
	fb_ton_quitt						: TON;
	fb_ton_taste_steuerung_ein				: TON;
	fb_ton_taste_steuerung_aus				: TON;
	fb_ton_taste_stoerung_quitt				: TON;
	fb_r_trig_quittieren					: R_TRIG;
	fb_state_entry						: ST_StateEntry;
	i32_fb_error_counter_gruppe1		: DINT := 0;
	i32_fb_error_counter_gruppe2		: DINT := 0;
	i32_fb_error_counter_gruppe3		: DINT := 0;
	i32_fb_error_counter_gruppe4		: DINT := 0;
	i32_com_error_counter_gruppe1		: DINT := 0;
	i32_com_error_counter_gruppe2		: DINT := 0;
	i32_com_error_counter_gruppe3		: DINT := 0;
	i32_com_error_counter_gruppe4		: DINT := 0;

	sm_steuerung_aus				: BOOL := FALSE;
	sm_not_halt_intern					: BOOL := FALSE;
	sm_not_halt_frontseite				: BOOL := FALSE;
	sm_not_halt_rueckseite			: BOOL := FALSE;
	sm_not_halt_bediengeraet			: BOOL := FALSE;
	sm_not_halt_extern				: BOOL := FALSE;
	sm_tuere_vorne_offen				: BOOL := FALSE;
	sm_tuere_hinten_offen				: BOOL := FALSE;
	sm_tuere_vorne_diskrepanz		: BOOL := FALSE;
	sm_tuere_hinten_diskrepanz		: BOOL := FALSE;
	sm_bestueckachse_sto			: BOOL := FALSE;
	sm_bestueckachse_sls			: BOOL := FALSE;
	sm_z_achse_sto					: BOOL := FALSE;
	sm_z_achse_sls					: BOOL := FALSE;
	sm_y_achse_sto					: BOOL := FALSE;
	sm_y_achse_sls					: BOOL := FALSE;
	sm_b_achse_sto					: BOOL := FALSE;
	sm_b_achse_sls					: BOOL := FALSE;
	sm_transport_achse_sto				: BOOL := FALSE;
	sm_transport_achse_sls			: BOOL := FALSE;

	bm_taste_steuerung_ein_verhaengt		: BOOL := FALSE;
	bm_taste_steuerung_aus_verhaengt		: BOOL := FALSE;
	bm_taste_stoerung_quitt_verhaengt		: BOOL := FALSE;

	sm_fehler_fb1_opmode					: BOOL := FALSE;
	sm_fehler_fb9_estop_nothalt_front			: BOOL := FALSE;
	sm_fehler_fb10_estop_nothalt_ext			: BOOL := FALSE;
	sm_fehler_fb15_edm_nothalt_ext				: BOOL := FALSE;
	sm_fehler_fb16_edm_nothalt_schuetz			: BOOL := FALSE;
	sm_fehler_fb17_edm_ventilinsel				: BOOL := FALSE;
	sm_fehler_fb28_edm_foerderband			: BOOL := FALSE;
	sm_fehler_fb30_estop_rueck				: BOOL := FALSE;
	sm_fehler_fb31_estop_bedien				: BOOL := FALSE;
	sm_fehler_fb35_mon_tuere_vo				: BOOL := FALSE;
	sm_fehler_fb36_mon_tuere_hi				: BOOL := FALSE;
	sm_fehler_fb37_mon_tuere_disk_vo			: BOOL := FALSE;
	sm_fehler_fb38_mon_tuere_disk_hi			: BOOL := FALSE;
	sm_fehler_fb39_mon_tuere_meld_vo			: BOOL := FALSE;
	sm_fehler_fb40_mon_tuere_meld_hi			: BOOL := FALSE;
	sm_not_halt_hublift_links					: BOOL := FALSE;

	a_quitt_pilz_hublift_links			AT %Q* : BOOL;

	a_lampe_quitt_schutztuere_vorne	AT %Q* : BOOL;
	a_lampe_quitt_schutztuere_hinten	AT %Q* : BOOL;

	(* Eingänge von Twinsafe FBs *)
	se_quittiertaste					AT %I* : BOOL;
	se_taste_steuerung_ein				AT %I* : BOOL;
	se_taste_steuerung_aus				AT %I* : BOOL;
	se_steuerung_ein					AT %I* : BOOL;
	se_ba_mit_bedingungen				AT %I* : BOOL;
	se_nothalt_gesamt_ok				AT %I* : BOOL;
	se_tuere_vorne_diskrepanz			AT %I* : BOOL;
	se_tuere_hinten_diskrepanz			AT %I* : BOOL;
	se_not_halt_intern					AT %I* : BOOL;
	se_not_halt_frontseite				AT %I* : BOOL;
	se_not_halt_rueckseite				AT %I* : BOOL;
	se_not_halt_bediengeraet			AT %I* : BOOL;
	se_not_halt_extern					AT %I* : BOOL;
	se_tuere_vorne_offen				AT %I* : BOOL;
	se_tuere_hinten_offen				AT %I* : BOOL;
	se_tuere_zustimm_vorne_offen		AT %I* : BOOL;
	se_tuere_zustimm_hinten_offen		AT %I* : BOOL;
	se_bestueckachse_sto				AT %I* : BOOL;
	se_bestueckachse_sls				AT %I* : BOOL;
	se_z_achse_sto					AT %I* : BOOL;
	se_z_achse_sls					AT %I* : BOOL;
	se_y_achse_sto					AT %I* : BOOL;
	se_y_achse_sls					AT %I* : BOOL;
	se_b_achse_sto					AT %I* : BOOL;
	se_b_achse_sls					AT %I* : BOOL;
	se_transport_achse_sto			AT %I* : BOOL;
	se_transport_achse_sls			AT %I* : BOOL;

	e_not_halt_hublift_links_ok				AT %I* : BOOL;	(* Not Halt OK Signal von Pilz Hublift links *)

	se_fehler_fb1_opmode						AT %I* : BOOL;
	se_fehler_fb9_estop_nothalt_front			AT %I* : BOOL;
	se_fehler_fb10_estop_nothalt_ext			AT %I* : BOOL;
	se_fehler_fb15_edm_nothalt_ext				AT %I* : BOOL;
	se_fehler_fb16_edm_nothalt_schuetz			AT %I* : BOOL;
	se_fehler_fb17_edm_ventilinsel				AT %I* : BOOL;
	se_fehler_fb28_edm_foerderband			AT %I* : BOOL;
	se_fehler_fb30_estop_rueck				AT %I* : BOOL;
	se_fehler_fb31_estop_bedien				AT %I* : BOOL;
	se_fehler_fb35_mon_tuere_vo				AT %I* : BOOL;
	se_fehler_fb36_mon_tuere_hi				AT %I* : BOOL;
	se_fehler_fb37_mon_tuere_disk_vo			AT %I* : BOOL;
	se_fehler_fb38_mon_tuere_disk_hi			AT %I* : BOOL;
	se_fehler_fb39_mon_tuere_meld_vo			AT %I* : BOOL;
	se_fehler_fb40_mon_tuere_meld_hi			AT %I* : BOOL;

	(* Betriebsarten *)
	sa_run_stop_gruppe1				AT %Q* : BOOL;
	sa_err_ack_gruppe1				AT %Q* : BOOL;
	se_fb_error_gruppe1				AT %I* : BOOL;
	se_com_error_gruppe1			AT %I* : BOOL;
	se_out_error_gruppe1				AT %I* : BOOL;
	(* Notaus *)
	sa_run_stop_gruppe2				AT %Q* : BOOL;
	sa_err_ack_gruppe2				AT %Q* : BOOL;
	se_fb_error_gruppe2				AT %I* : BOOL;
	se_com_error_gruppe2			AT %I* : BOOL;
	se_out_error_gruppe2				AT %I* : BOOL;
	(* Türen *)
	sa_run_stop_gruppe3				AT %Q* : BOOL;
	sa_err_ack_gruppe3				AT %Q* : BOOL;
	se_fb_error_gruppe3				AT %I* : BOOL;
	se_com_error_gruppe3			AT %I* : BOOL;
	se_out_error_gruppe3				AT %I* : BOOL;
	(* Safety AX5000 *)
	sa_run_stop_gruppe4				AT %Q* : BOOL;
	sa_err_ack_gruppe4				AT %Q* : BOOL;
	se_fb_error_gruppe4				AT %I* : BOOL;
	se_com_error_gruppe4			AT %I* : BOOL;
	se_out_error_gruppe4				AT %I* : BOOL;
END_VAR
(* Zeiten *)
fb_ton_wz(IN:= , PT:= T#100ms, Q=>  , ET=> );
fb_ton_quitt(IN:= , PT:= t#20ms, Q=> , ET=> );
fb_ton_taste_steuerung_ein(IN:= se_taste_steuerung_ein, PT:= t#60s, Q=> bm_taste_steuerung_ein_verhaengt, ET=> );
fb_ton_taste_steuerung_aus(IN:= NOT se_taste_steuerung_aus, PT:= t#60s, Q=> bm_taste_steuerung_aus_verhaengt, ET=> );
fb_ton_taste_stoerung_quitt(IN:= se_quittiertaste, PT:= t#60s, Q=> bm_taste_stoerung_quitt_verhaengt, ET=> );

(* Flanken *)
fb_r_trig_quittieren(CLK:= visu.b_quittieren, Q=> );

(* Startsignal für die Safety-Gruppen *)
sa_run_stop_gruppe1 := TRUE;
sa_run_stop_gruppe2 := TRUE;
sa_run_stop_gruppe3 := TRUE;
sa_run_stop_gruppe4 := TRUE;

(* Automatische Quittierung von Errors in den TwinSafe-Gruppen *)
ack_step(
	i16_next_step:= ,
	i16_pos:= 1,
	s_debugtext:= ,
	E=> ,
	X=> ,
	i16_step=> ,
	i16_last_step=> );

CASE ack_step.i16_step OF
	0:	(* Nach Startup automatische Quittierung von FB- und COM-Fehlern *)
		IF 	se_fb_error_gruppe1 OR
			se_com_error_gruppe1 OR
			se_fb_error_gruppe2 OR
			se_com_error_gruppe2 OR
			se_fb_error_gruppe3 OR
			se_com_error_gruppe3 OR
			se_fb_error_gruppe4 OR
			se_com_error_gruppe4
			THEN
				sa_err_ack_gruppe1 := FALSE;
				sa_err_ack_gruppe2 := FALSE;
				sa_err_ack_gruppe3 := FALSE;
				sa_err_ack_gruppe4 := FALSE;
				fb_ton_wz.IN := TRUE;
				IF fb_ton_wz.Q THEN
					fb_ton_wz.IN := FALSE;
					ack_step.i16_next_step := 10;
				END_IF
		END_IF

	10:
		sa_err_ack_gruppe1 := TRUE;
		sa_err_ack_gruppe2 := TRUE;
		sa_err_ack_gruppe3 := TRUE;
		sa_err_ack_gruppe4 := TRUE;
		fb_ton_wz.IN := TRUE;
		IF fb_ton_wz.Q THEN
			fb_ton_wz.IN := FALSE;
			ack_step.i16_next_step := 20;
		END_IF

	20:
		sa_err_ack_gruppe1 := FALSE;
		sa_err_ack_gruppe2 := FALSE;
		sa_err_ack_gruppe3 := FALSE;
		sa_err_ack_gruppe4 := FALSE;
		fb_ton_wz.IN := TRUE;
		IF fb_ton_wz.Q THEN
			fb_ton_wz.IN := FALSE;
			ack_step.i16_next_step := 100;
		END_IF

	100:	(* FB- und COM-Fehler  *)
		IF 	se_fb_error_gruppe1 OR
			se_com_error_gruppe1 OR
			se_fb_error_gruppe2 OR
			se_com_error_gruppe2 OR
			se_fb_error_gruppe3 OR
			se_com_error_gruppe3 OR
			se_fb_error_gruppe4 OR
			se_com_error_gruppe4
			THEN
				sa_err_ack_gruppe1 := FALSE;
				sa_err_ack_gruppe2 := FALSE;
				sa_err_ack_gruppe3 := FALSE;
				sa_err_ack_gruppe4 := FALSE;
				ack_step.i16_next_step := 110;
		END_IF

	110:
		IF ack_step.E THEN
			IF se_fb_error_gruppe1 THEN
				i32_fb_error_counter_gruppe1 := i32_fb_error_counter_gruppe1 + 1;
			END_IF
			IF se_fb_error_gruppe2 THEN
				i32_fb_error_counter_gruppe2 := i32_fb_error_counter_gruppe2 + 1;
			END_IF
			IF se_fb_error_gruppe3 THEN
				i32_fb_error_counter_gruppe3 := i32_fb_error_counter_gruppe3 + 1;
			END_IF
			IF se_fb_error_gruppe4 THEN
				i32_fb_error_counter_gruppe4 := i32_fb_error_counter_gruppe4 + 1;
			END_IF
			IF se_com_error_gruppe1 THEN
				i32_com_error_counter_gruppe1 := i32_com_error_counter_gruppe1 + 1;
			END_IF
			IF se_com_error_gruppe2 THEN
				i32_com_error_counter_gruppe2 := i32_com_error_counter_gruppe2 + 1;
			END_IF
			IF se_com_error_gruppe3 THEN
				i32_com_error_counter_gruppe3 := i32_com_error_counter_gruppe3 + 1;
			END_IF
			IF se_com_error_gruppe4 THEN
				i32_com_error_counter_gruppe4 := i32_com_error_counter_gruppe4 + 1;
			END_IF
		END_IF
		ack_step.i16_next_step := 120;

	120:
		sa_err_ack_gruppe1 := TRUE;
		sa_err_ack_gruppe2 := TRUE;
		sa_err_ack_gruppe3 := TRUE;
		sa_err_ack_gruppe4 := TRUE;
		fb_ton_wz.IN := TRUE;
		IF fb_ton_wz.Q THEN
			fb_ton_wz.IN := FALSE;
			ack_step.i16_next_step := 130;
		END_IF

	130:
		sa_err_ack_gruppe1 := FALSE;
		sa_err_ack_gruppe2 := FALSE;
		sa_err_ack_gruppe3 := FALSE;
		sa_err_ack_gruppe4 := FALSE;
		fb_ton_wz.IN := TRUE;
		IF fb_ton_wz.Q THEN
			fb_ton_wz.IN := FALSE;
			ack_step.i16_next_step := 100;
		END_IF
END_CASE

ack_step(
	i16_next_step:= ,
	i16_pos:= 2,
	s_debugtext:= ,
	E=> ,
	X=> , 
	i16_step=> ,
	i16_last_step=> );


(* Lampen für Schutztüren *)
a_lampe_quitt_schutztuere_hinten := NOT se_tuere_hinten_offen;
a_lampe_quitt_schutztuere_vorne := 	NOT se_tuere_vorne_offen OR
								NOT se_tuere_hinten_offen OR
								NOT se_not_halt_intern;

(* Quittierung Pilz Hublift links *)
a_quitt_pilz_hublift_links := se_quittiertaste;

(* ======================================Schrittkette======================================== *)
fb_state_entry(
	i16_next_step:= ,
	i16_pos:= 1,
	s_debugtext:= ,
	E=> ,
	X=> ,
	i16_step=> ,
	i16_last_step=> );

CASE fb_state_entry.i16_step OF
(*=======================================================*)
	INIT_OBJ:
		IF	st_config.b_config_fertig AND
			NOT se_fb_error_gruppe1 AND
			NOT se_com_error_gruppe1 AND
			NOT se_fb_error_gruppe2 AND
			NOT se_com_error_gruppe2 AND
			NOT se_fb_error_gruppe3 AND
			NOT se_com_error_gruppe3 AND
			NOT se_fb_error_gruppe4 AND
			NOT se_com_error_gruppe4
			THEN
				fb_state_entry.i16_next_step := INIT;
		END_IF

(*=======================================================*)
	INIT:
		st_ctrl_out.b_fehler := FALSE;
		st_ctrl_out.b_bereit := FALSE;
		fb_ton_quitt.IN := FALSE;
		sm_steuerung_aus := FALSE;
		sm_not_halt_intern := FALSE;
		sm_not_halt_frontseite := FALSE;
		sm_not_halt_rueckseite := FALSE;
		sm_not_halt_bediengeraet := FALSE;
		sm_not_halt_extern := FALSE;
		sm_tuere_vorne_offen := FALSE;
		sm_tuere_hinten_offen := FALSE;
		sm_tuere_vorne_diskrepanz := FALSE;
		sm_tuere_hinten_diskrepanz := FALSE;
		sm_bestueckachse_sto := FALSE;
		sm_bestueckachse_sls := FALSE;
		sm_z_achse_sto := FALSE;
		sm_z_achse_sls := FALSE;
		sm_y_achse_sto := FALSE;
		sm_y_achse_sls := FALSE;
		sm_b_achse_sto := FALSE;
		sm_b_achse_sls := FALSE;
		sm_transport_achse_sto := FALSE;
		sm_transport_achse_sls := FALSE;
		sm_fehler_fb1_opmode := FALSE;
		sm_fehler_fb9_estop_nothalt_front := FALSE;
		sm_fehler_fb10_estop_nothalt_ext := FALSE;
		sm_fehler_fb15_edm_nothalt_ext	 := FALSE;
		sm_fehler_fb16_edm_nothalt_schuetz := FALSE;
		sm_fehler_fb17_edm_ventilinsel := FALSE;
		sm_fehler_fb28_edm_foerderband := FALSE;
		sm_fehler_fb30_estop_rueck := FALSE;
		sm_fehler_fb31_estop_bedien := FALSE;
		sm_fehler_fb35_mon_tuere_vo := FALSE;
		sm_fehler_fb36_mon_tuere_hi := FALSE;
		sm_fehler_fb37_mon_tuere_disk_vo := FALSE;
		sm_fehler_fb38_mon_tuere_disk_hi := FALSE;
		sm_fehler_fb39_mon_tuere_meld_vo := FALSE;
		sm_fehler_fb40_mon_tuere_meld_hi := FALSE;
		sm_not_halt_hublift_links := FALSE;

		(*-----------------------Weiterschaltbedingungen----------------------------*)
		fb_state_entry.i16_next_step := BEREIT;

(*=======================================================*)
	BEREIT:
		IF fb_state_entry.E THEN
			st_ctrl_out.b_bereit := TRUE;
		END_IF

		(* Hinweis: SLS der Achsen endet immer bei STO, deshalb wird nur STO abgefragt *)
		CASE gst_datensatz.st_md.i16_typ_zelle OF
			KEINE_ZELLE:
				;

			BESTUECKZELLE_1700, RASTERFOLIE:
				IF	se_steuerung_ein AND
					se_not_halt_intern AND
					se_not_halt_extern AND
					se_tuere_zustimm_vorne_offen AND
					se_tuere_zustimm_hinten_offen AND
					(*se_tuere_vorne_offen AND
					se_tuere_hinten_offen AND*)
					NOT se_bestueckachse_sto AND
					NOT se_z_achse_sto AND
					NOT se_y_achse_sto AND
					NOT se_tuere_vorne_diskrepanz AND
					NOT se_tuere_hinten_diskrepanz AND
					(e_not_halt_hublift_links_ok OR NOT gst_datensatz.st_md.b_hublift_links_aktiv)
					THEN
						;
				ELSE
					fb_state_entry.i16_next_step := FEHLER;
				END_IF

			BESTUECKZELLE_1720:
				IF	se_steuerung_ein AND
					se_not_halt_intern AND
					se_not_halt_extern AND
					se_tuere_zustimm_vorne_offen AND
					se_tuere_zustimm_hinten_offen AND
					(*se_tuere_vorne_offen AND
					se_tuere_hinten_offen AND*)
					NOT se_bestueckachse_sto AND
					NOT se_z_achse_sto AND
					NOT se_tuere_vorne_diskrepanz AND
					NOT se_tuere_hinten_diskrepanz AND
					(e_not_halt_hublift_links_ok OR NOT gst_datensatz.st_md.b_hublift_links_aktiv)
					THEN
						;
				ELSE
					fb_state_entry.i16_next_step := FEHLER;
				END_IF
		END_CASE

(*=======================================================*)
	FEHLER:
		IF fb_state_entry.E THEN
			st_ctrl_out.b_fehler := TRUE;
			fb_ton_quitt.IN := FALSE;
		END_IF

		(* Gruppe NOT-AUS *)
		sm_not_halt_frontseite := NOT se_not_halt_frontseite;
		sm_not_halt_rueckseite := NOT se_not_halt_rueckseite;
		sm_not_halt_bediengeraet := NOT se_not_halt_bediengeraet;
		sm_steuerung_aus := NOT se_steuerung_ein AND se_not_halt_frontseite AND se_not_halt_rueckseite AND se_not_halt_bediengeraet AND se_tuere_vorne_offen AND se_tuere_hinten_offen;
		sm_not_halt_extern := NOT se_not_halt_extern;

		IF se_steuerung_ein AND se_not_halt_frontseite AND se_not_halt_rueckseite AND se_not_halt_bediengeraet THEN
			(* Gruppe Achsen *)
			sm_bestueckachse_sto := 	se_bestueckachse_sto AND
									(gst_datensatz.st_md.i16_typ_zelle = BESTUECKZELLE_1700 OR gst_datensatz.st_md.i16_typ_zelle = BESTUECKZELLE_1720);
			sm_z_achse_sto := se_z_achse_sto;
			sm_y_achse_sto := se_y_achse_sto AND
								gst_datensatz.st_md.i16_typ_zelle = BESTUECKZELLE_1700 ;
			sm_b_achse_sto := se_b_achse_sto AND
							(gst_datensatz.st_wkz.i16_typ_bandeinzug = SERVO);
			sm_transport_achse_sto := se_transport_achse_sto AND
							(gst_datensatz.st_md.b_anwahl_transport_achse);
		END_IF

		(* Gruppe Schutzeinrichtungen *)
		(* Schutztüren Bestückautomat vorne *)
		sm_tuere_vorne_offen :=  NOT se_tuere_vorne_offen;
		sm_tuere_vorne_diskrepanz := se_tuere_vorne_diskrepanz;
		(* Schutztüren Bestückautomat hinten *)
		sm_tuere_hinten_offen := NOT se_tuere_hinten_offen;
		sm_tuere_hinten_diskrepanz := se_tuere_hinten_diskrepanz;

		(* SAFETY- FB-Fehler *)
		sm_fehler_fb1_opmode := se_fehler_fb1_opmode;
		sm_fehler_fb9_estop_nothalt_front := se_fehler_fb9_estop_nothalt_front;
		sm_fehler_fb10_estop_nothalt_ext := se_fehler_fb10_estop_nothalt_ext;
		sm_fehler_fb15_edm_nothalt_ext := se_fehler_fb15_edm_nothalt_ext;
		sm_fehler_fb16_edm_nothalt_schuetz := se_fehler_fb16_edm_nothalt_schuetz;
		sm_fehler_fb17_edm_ventilinsel := se_fehler_fb17_edm_ventilinsel;
		sm_fehler_fb28_edm_foerderband := se_fehler_fb28_edm_foerderband;
		sm_fehler_fb30_estop_rueck := se_fehler_fb30_estop_rueck;
		sm_fehler_fb31_estop_bedien := se_fehler_fb31_estop_bedien;
		sm_fehler_fb35_mon_tuere_vo := se_fehler_fb35_mon_tuere_vo;
		sm_fehler_fb36_mon_tuere_hi := se_fehler_fb36_mon_tuere_hi;
		sm_fehler_fb37_mon_tuere_disk_vo := se_fehler_fb37_mon_tuere_disk_vo;
		sm_fehler_fb38_mon_tuere_disk_hi := se_fehler_fb38_mon_tuere_disk_hi;
		sm_fehler_fb39_mon_tuere_meld_vo := se_fehler_fb39_mon_tuere_meld_vo;
		sm_fehler_fb40_mon_tuere_meld_hi := se_fehler_fb40_mon_tuere_meld_hi;

		IF gst_datensatz.st_md.b_hublift_links_aktiv THEN
			sm_not_halt_hublift_links := NOT e_not_halt_hublift_links_ok;
		END_IF

		(*-----------------------Weiterschaltbedingungen----------------------------*)
		IF st_ctrl_in.b_quitt AND NOT fb_state_entry.E THEN
			st_ctrl_out.b_fehler := FALSE;
			fb_ton_quitt.IN := TRUE;
		END_IF

		IF fb_ton_quitt.Q THEN
			fb_ton_quitt.IN := FALSE;
			fb_state_entry.i16_next_step := INIT;
		END_IF
END_CASE

fb_state_entry(
	i16_next_step:= ,
	i16_pos:= 2,
	s_debugtext:= ,
	E=> ,
	X=> , 
	i16_step=> ,
	i16_last_step=> );

IF st_config.b_config_fertig THEN
	(* Fehlermeldungen und Betriebsmeldungen ab dem Startindex in die globalen Meldungsarrays schreiben *)
	garr_stoermeldungen[st_config.i16_meld_startindex + 0] := sm_steuerung_aus;
	garr_stoermeldungen[st_config.i16_meld_startindex + 1] := sm_not_halt_intern;
	garr_stoermeldungen[st_config.i16_meld_startindex + 2] := sm_not_halt_extern;
	garr_stoermeldungen[st_config.i16_meld_startindex + 3] := sm_tuere_vorne_offen;
	garr_stoermeldungen[st_config.i16_meld_startindex + 4] := sm_tuere_hinten_offen;
	garr_stoermeldungen[st_config.i16_meld_startindex + 5] := sm_tuere_vorne_diskrepanz;
	garr_stoermeldungen[st_config.i16_meld_startindex + 6] := sm_tuere_hinten_diskrepanz;
	garr_stoermeldungen[st_config.i16_meld_startindex + 7] := sm_bestueckachse_sto;
	garr_stoermeldungen[st_config.i16_meld_startindex + 8] := sm_bestueckachse_sls;
	garr_stoermeldungen[st_config.i16_meld_startindex + 9] := sm_z_achse_sto;
	garr_stoermeldungen[st_config.i16_meld_startindex + 10] := sm_z_achse_sls;
	garr_stoermeldungen[st_config.i16_meld_startindex + 11] := sm_y_achse_sto;
	garr_stoermeldungen[st_config.i16_meld_startindex + 12] := sm_y_achse_sls;
	garr_stoermeldungen[st_config.i16_meld_startindex + 13] := sm_not_halt_frontseite;
	garr_stoermeldungen[st_config.i16_meld_startindex + 14] := sm_not_halt_rueckseite;
	garr_stoermeldungen[st_config.i16_meld_startindex + 15] := sm_not_halt_bediengeraet;
	garr_stoermeldungen[st_config.i16_meld_startindex + 16] := sm_b_achse_sto;
	garr_stoermeldungen[st_config.i16_meld_startindex + 17] := sm_b_achse_sls;
	garr_stoermeldungen[st_config.i16_meld_startindex + 18] := sm_transport_achse_sto;
	garr_stoermeldungen[st_config.i16_meld_startindex + 19] := sm_transport_achse_sls;
	garr_stoermeldungen[st_config.i16_meld_startindex + 20] := sm_fehler_fb1_opmode;
	garr_stoermeldungen[st_config.i16_meld_startindex + 21] := sm_fehler_fb9_estop_nothalt_front;
	garr_stoermeldungen[st_config.i16_meld_startindex + 22] := sm_fehler_fb10_estop_nothalt_ext;
	garr_stoermeldungen[st_config.i16_meld_startindex + 23] := sm_fehler_fb15_edm_nothalt_ext	;
	garr_stoermeldungen[st_config.i16_meld_startindex + 24] := sm_fehler_fb16_edm_nothalt_schuetz;
	garr_stoermeldungen[st_config.i16_meld_startindex + 25] := sm_fehler_fb17_edm_ventilinsel;
	garr_stoermeldungen[st_config.i16_meld_startindex + 26] := sm_fehler_fb28_edm_foerderband;
	garr_stoermeldungen[st_config.i16_meld_startindex + 27] := sm_fehler_fb30_estop_rueck;
	garr_stoermeldungen[st_config.i16_meld_startindex + 28] := sm_fehler_fb31_estop_bedien;
	garr_stoermeldungen[st_config.i16_meld_startindex + 29] := sm_fehler_fb35_mon_tuere_vo;
	garr_stoermeldungen[st_config.i16_meld_startindex + 30] := sm_fehler_fb36_mon_tuere_hi;
	garr_stoermeldungen[st_config.i16_meld_startindex + 31] := sm_fehler_fb37_mon_tuere_disk_vo;
	garr_stoermeldungen[st_config.i16_meld_startindex + 32] := sm_fehler_fb38_mon_tuere_disk_hi;
	garr_stoermeldungen[st_config.i16_meld_startindex + 33] := sm_fehler_fb39_mon_tuere_meld_vo;
	garr_stoermeldungen[st_config.i16_meld_startindex + 34] := sm_fehler_fb40_mon_tuere_meld_hi;
	garr_stoermeldungen[st_config.i16_meld_startindex + 35] := sm_not_halt_hublift_links;
	garr_stoermeldungen[st_config.i16_meld_startindex + 36] := FALSE;
	garr_stoermeldungen[st_config.i16_meld_startindex + 37] := FALSE;
	garr_stoermeldungen[st_config.i16_meld_startindex + 38] := FALSE;
	garr_stoermeldungen[st_config.i16_meld_startindex + 39] := FALSE;

	garr_betriebsmeldungen[st_config.i16_meld_startindex + 0] := bm_taste_steuerung_ein_verhaengt;
	garr_betriebsmeldungen[st_config.i16_meld_startindex + 1] := bm_taste_steuerung_aus_verhaengt;
	garr_betriebsmeldungen[st_config.i16_meld_startindex + 2] := bm_taste_stoerung_quitt_verhaengt;
	garr_betriebsmeldungen[st_config.i16_meld_startindex + 3] := FALSE;
	garr_betriebsmeldungen[st_config.i16_meld_startindex + 4] := FALSE;
	garr_betriebsmeldungen[st_config.i16_meld_startindex + 5] := FALSE;
	garr_betriebsmeldungen[st_config.i16_meld_startindex + 6] := FALSE;
	garr_betriebsmeldungen[st_config.i16_meld_startindex + 7] := FALSE;
	garr_betriebsmeldungen[st_config.i16_meld_startindex + 8] := FALSE;
	garr_betriebsmeldungen[st_config.i16_meld_startindex + 9] := FALSE;
	garr_betriebsmeldungen[st_config.i16_meld_startindex + 10] := FALSE;
	garr_betriebsmeldungen[st_config.i16_meld_startindex + 11] := FALSE;
	garr_betriebsmeldungen[st_config.i16_meld_startindex + 12] := FALSE;
	garr_betriebsmeldungen[st_config.i16_meld_startindex + 13] := FALSE;
	garr_betriebsmeldungen[st_config.i16_meld_startindex + 14] := FALSE;
	garr_betriebsmeldungen[st_config.i16_meld_startindex + 15] := FALSE;
	garr_betriebsmeldungen[st_config.i16_meld_startindex + 16] := FALSE;
	garr_betriebsmeldungen[st_config.i16_meld_startindex + 17] := FALSE;
	garr_betriebsmeldungen[st_config.i16_meld_startindex + 18] := FALSE;
	garr_betriebsmeldungen[st_config.i16_meld_startindex + 19] := FALSE;
END_IF
END_PROGRAM

(* POU EPT Lib/Funktionen/F_Vergleich_LReal, ST *)
FUNCTION F_Vergleich_LReal : BOOL
VAR_INPUT
	lr_wert			: LREAL;
	lr_vergleichswert	: LREAL;
END_VAR
VAR
	lr_toleranz		: LREAL := 0.02;
END_VAR
IF ABS(lr_wert - lr_vergleichswert) < lr_toleranz THEN
	F_Vergleich_LReal := TRUE;
ELSE
	F_Vergleich_LReal := FALSE;
END_IF
END_FUNCTION

(* POU Gemeinsamkeiten17xx/Wartung/ST_Wartung, ST *)
PROGRAM ST_Wartung
VAR_INPUT
	st_config								: struct_config;
	st_ctrl_in								: struct_ctrl_in;
END_VAR
VAR_IN_OUT
	i16_auftrag							: enum_wartung_auftrag;
END_VAR
VAR_OUTPUT
	st_ctrl_out								: struct_ctrl_out;
END_VAR
VAR
	(*Bausteinaufrufe*)
	fb_state_entry					: ST_StateEntry;
	fb_ton_quitt						: TON;
	fb_xml_srv_read					: FB_XmlSrvReadByName;
	fb_xml_srv_write					: FB_XmlSrvWriteByName;
	fbFindFiles						: FB_EnumFindFileList;
	file								: ST_FindFileEntry;
	FB_GetHostName				: FB_GetHostName;
	fb_nt_start_process				: NT_StartProcess;

	(*Flanken*)
	fb_r_trig_autosafe				: R_TRIG;
	fb_r_trig_reset_wkz			: R_TRIG;

	(*Zeiten*)
	fb_ton_wz									: TON;
	fb_ton_wz_wartung				: TON;
	fb_ton_end								: TON;
	fb_ton_autosafe					: TON;


	(* Dateiname *)
	sFileName_md							: STRING;
	sFileName_wkz						: STRING;
	sHelpName							: STRING;
	sHelpPos							: INT;

	(* Dateipfad *)
	sPathName								: STRING;

	(* Temporäre Variable *)
	b_init											: BOOL;
	b_lesen_komplett					: BOOL := TRUE;
	b_datei_vorhanden				: BOOL;
	b_auto_speichern_auf_server		: BOOL ;
	nErrId											: UDINT;
	sm_fehler_schreiben_Wartungsprotokoll			: BOOL;
	sm_fehler_lesen_Wartungsprotokoll					: BOOL;
	sm_fehler_speichern_Wartungsprotokoll			: BOOL;

	s_aktuelles_wkz_copy											: STRING;
	i																					: INT:=0;

	st_wartungsprotokoll_md_copy							: struct_Wartungsprotokoll;
	st_wartungsprotokoll_wkz_copy							: struct_Wartungsprotokoll;
	i32_bestueckhubzaehler_md_copy					: UDINT := 0;
	i32_bestueckhubzaehler_wkz_copy				: UDINT := 0;
END_VAR

VAR CONSTANT
	st_wartungsprotokoll_leer			: struct_Wartungsprotokoll;
	s_wartung_path_wkz					: STRING(50):='D:\BBgen\Wartung\Werkzeug\';
	s_wartung_path_md						: STRING(50):='D:\BBgen\Wartung\Maschine\';
	s_Trennstelle									: STRING(2):='#';
END_VAR
FileName_erstellen ();
fb_Aufrufe ();
auto_speichern_laden ();

IF NOT b_init AND gst_datensatz.st_md.s_aktuelles_wkz <>''  THEN
	i16_auftrag:= LESE_WARTUNGSPROTOKOLL_KOMPLETT;
	s_aktuelles_wkz_copy:=gst_datensatz.st_md.s_aktuelles_wkz;
	i32_bestueckhubzaehler_md_copy:=gst_datensatz.st_md.i32_bestueckhubzaehler;
	FB_GetHostName.bExecute := TRUE;
	b_init := TRUE;
ELSIF b_init AND gst_datensatz.st_md.s_aktuelles_wkz <> s_aktuelles_wkz_copy AND gi16_maschinenstatusinfo <> STATUS_MASCHINE_ARBEITET THEN
	i16_auftrag:=LESE_WARTUNGSPROTOKOLL_WKZ;
	i32_bestueckhubzaehler_md_copy:=gst_datensatz.st_md.i32_bestueckhubzaehler;
	s_aktuelles_wkz_copy:=gst_datensatz.st_md.s_aktuelles_wkz;
ELSE
	Zaehler();
END_IF


(*Zellennummer aus dem Computernamen filtern*)
sHelpName := FB_GetHostName.sHostName;
sHelpPos := FIND(sHelpName,'-');
sHelpName := DELETE(sHelpName,sHelpPos,1);
sHelpPos := FIND(sHelpName,'-');
sHelpName := LEFT(sHelpName,sHelpPos-1);
sHelpName := CONCAT('T#',sHelpName);
sHelpName := CONCAT(sHelpName,'s');

(* Flanken *)
fb_r_trig_reset_wkz(CLK:= visu.b_reset_wartung_wkz, Q=> );
fb_r_trig_autosafe(CLK:= gstr_uhrzeit = '01:00:00', Q=> );
fb_ton_autosafe(IN:= , PT:= STRING_TO_TIME(sHelpName), Q=> , ET=> );

IF fb_r_trig_autosafe.Q THEN
	fb_ton_autosafe.IN := TRUE;
END_IF

(*Um 1 Uhr + Zellennummer in Sek. früh werden die Wartungsprotokolle an den Server geschickt*)
IF fb_ton_autosafe.Q THEN
	b_auto_speichern_auf_server := TRUE;
	fb_ton_autosafe.IN := FALSE;
END_IF

IF b_auto_speichern_auf_server AND i16_auftrag = KEIN_WARTUNG_AUFTRAG THEN
	b_auto_speichern_auf_server := FALSE;
	IF visu.s_akt_sprache = 'de' THEN
		i16_auftrag:=SPEICHERN_WARTUNGSPROTOKOLL;
	END_IF
END_IF


(*
IF visu.b_reset_wartung_maschine THEN
	gst_datensatz.st_md.produzierte_stecker := 0;
END_IF
*)

(*Zeiten*)
fb_ton_wz(IN:= , PT:= , Q=> , ET=> );
fb_ton_quitt(IN:= , PT:= t#100ms, Q=> , ET=> );

(* ======================================Schrittkette======================================== *)
fb_state_entry(i16_pos:= 1);


CASE fb_state_entry.i16_step OF
(*=======================================================*)
	INIT_OBJ:
		(*-----------------------Weiterschaltbedingungen----------------------------*)
		IF FB_GetHostName.bBusy OR FB_GetHostName.sHostName <> '' THEN
			fb_state_entry.i16_next_step := 5;
		END_IF

		IF fb_state_entry.X THEN
			FB_GetHostName.bExecute := FALSE;
		END_IF

(*=======================================================*)
	5:
		(*-----------------------Weiterschaltbedingungen----------------------------*)
		IF NOT FB_GetHostName.bBusy THEN
			fb_state_entry.i16_next_step := INIT;
		END_IF

(*=======================================================*)
	INIT:	(*initialisieren*)
		st_ctrl_out.b_fehler := FALSE;
		st_ctrl_out.b_bereit := FALSE;
		st_ctrl_out.b_busy := FALSE;
		st_ctrl_out.b_fertig := FALSE;
		sm_fehler_schreiben_Wartungsprotokoll	 := FALSE;
		sm_fehler_lesen_Wartungsprotokoll	:= FALSE;
		sm_fehler_speichern_Wartungsprotokoll := FALSE;
		fbFindFiles.bExecute := FALSE;
		fb_xml_srv_write.bExecute := FALSE;
		fb_xml_srv_read.bExecute := FALSE;
		fb_ton_wz.IN := FALSE;

		fb_nt_start_process.START := FALSE;
		fbFindFiles.eCmd := 0;
		nErrId := 0;
		sPathName := '';
		b_datei_vorhanden := FALSE;
		fb_xml_srv_write.sSymName := '';
		fb_xml_srv_write.sXPath := '';

		(*-----------------------Weiterschaltbedingungen----------------------------*)
		fb_state_entry.i16_next_step:=BEREIT;


(*=======================================================*)
	BEREIT:(*Start*)
		IF 	fb_state_entry.E THEN
			st_ctrl_out.b_bereit := TRUE;
		END_IF

		CASE i16_auftrag OF
			LESE_WARTUNGSPROTOKOLL_KOMPLETT:
				b_lesen_komplett := TRUE;
				fb_state_entry.i16_next_step:=110;

			LESE_WARTUNGSPROTOKOLL_WKZ:
				fb_state_entry.i16_next_step:=110;

			LESE_WARTUNGSPROTOKOLL_MD:
				fb_state_entry.i16_next_step:=150;

			SCHREIBE_WARTUNGSPROTOKOLL_WKZ:
				fb_state_entry.i16_next_step:=200;

			SCHREIBE_WARTUNGSPROTOKOLL_MD:
				fb_state_entry.i16_next_step:=250;

			SPEICHERN_WARTUNGSPROTOKOLL:
				fb_state_entry.i16_next_step:=300;

			SCHREIBE_WARTUNGSPROTOKOLL_WKZ_RESET:
				fb_state_entry.i16_next_step:=400;
		END_CASE

		IF fb_state_entry.X THEN
			st_ctrl_out.b_bereit := FALSE;
			st_ctrl_out.b_fertig := FALSE;
			st_ctrl_out.b_busy := TRUE;
		END_IF

(*=======================================================*)
	110:(*Prüfe, ob Werkzeug Datei vorhanden ist*)
		IF fb_state_entry.E THEN
			sPathName := CONCAT(s_wartung_path_wkz,sFileName_wkz);
			sPathName:=CONCAT(sPathName,'.xml');
			(*Erste Datei im Verzeichnis kontrollieren*)
			IF fb_state_entry.i16_last_step <> 120 THEN
				fbFindFiles.eCmd := 0;
			(*Dateien im Verzeichnis durchzählen*)
			ELSE
				fbFindFiles.eCmd := 1;
			END_IF
			fbFindFiles.bExecute := TRUE;
		END_IF

		(*-----------------------Weiterschaltbedingungen----------------------------*)
		IF fbFindFiles.bBusy THEN
			fb_state_entry.i16_next_step:=120;
		END_IF

		IF fb_state_entry.X THEN
			fbFindFiles.bExecute := FALSE;
		END_IF

(*=======================================================*)
	120:(*Prüfe, ob Werkzeug Datei vorhanden ist*)
		(*-----------------------Weiterschaltbedingungen----------------------------*)
		(*letzte Datei im Verzeichnis erreicht*)
		IF fbFindFiles.bEOE AND NOT fbFindFiles.bBusy AND NOT fbFindFiles.bError  THEN
			IF fbFindFiles.nFindFiles <> 0 OR b_datei_vorhanden  THEN
				(*Datei vorhanden -> muss eingelesen werden*)
				fb_state_entry.i16_next_step:=130;
			ELSE
				(*Datei noch nicht vorhanden -> kann nicht eingelesen werden*)
				i32_bestueckhubzaehler_wkz_copy := 0;
				IF b_lesen_komplett THEN
					fb_state_entry.i16_next_step:=150;
				ELSE
					fb_state_entry.i16_next_step := 999;
				END_IF
			END_IF
		(*Datei wurde im Verzeichnis gefunden*)
		ELSIF NOT fbFindFiles.bBusy AND NOT fbFindFiles.bError  THEN
			IF fbFindFiles.nFindFiles <> 0  THEN
				(*Datei vorhanden -> muss eingelesen werden*)
				b_datei_vorhanden := TRUE;
				fb_state_entry.i16_next_step := 110;
			END_IF
		ELSIF fbFindFiles.bError THEN
			nErrId := fbFindFiles.nErrID;
			sm_fehler_lesen_Wartungsprotokoll := TRUE;
			fb_state_entry.i16_next_step:=FEHLER;
		END_IF

(*=======================================================*)
	130:	(* Lesen Werkzeug Wartungsprotokoll *)
		IF fb_state_entry.E THEN
			b_datei_vorhanden := FALSE;
			sPathName := CONCAT(s_wartung_path_wkz,sFileName_wkz);
			sPathName:=CONCAT(sPathName,'.xml');
			fb_xml_srv_read.sSymName := '.gst_datensatz.st_wartungsprotokoll.st_wartung_wkz';
			fb_xml_srv_read.sXPath := '/root/gst_datensatz.st_wartungsprotokoll.st_wartung_wkz';
			fb_xml_srv_read.bExecute:= TRUE;
		END_IF

		(*-----------------------Weiterschaltbedingungen----------------------------*)
		IF fb_xml_srv_read.bBusy THEN
			fb_state_entry.i16_next_step := 140;
		END_IF

		IF fb_state_entry.X THEN
			fb_xml_srv_read.bExecute:= FALSE;
		END_IF

(*=======================================================*)
	140:
		(*-----------------------Weiterschaltbedingungen----------------------------*)
		(*Lesen erfolgreich*)
		IF NOT fb_xml_srv_read.bError AND NOT fb_xml_srv_read.bBusy AND NOT b_lesen_komplett THEN
			i32_bestueckhubzaehler_wkz_copy := gst_datensatz.st_wartungsprotokoll.st_wartung_wkz.hubzaehler;
			fb_state_entry.i16_next_step := 999;
		ELSIF NOT fb_xml_srv_read.bError AND NOT fb_xml_srv_read.bBusy AND b_lesen_komplett THEN
			i32_bestueckhubzaehler_wkz_copy := gst_datensatz.st_wartungsprotokoll.st_wartung_wkz.hubzaehler;
			fb_state_entry.i16_next_step := 150;
		ELSIF fb_xml_srv_read.bError THEN
			nErrId:=fb_xml_srv_read.nErrId;
			sm_fehler_lesen_Wartungsprotokoll:=TRUE;
			fb_state_entry.i16_next_step := FEHLER;
		END_IF

(*=======================================================*)
	150:(*Prüfe, ob Maschinen Datei vorhanden ist*)
		IF fb_state_entry.E THEN
			sPathName := CONCAT(s_wartung_path_md,sFileName_md);
			(*Erste Datei im Verzeichnis kontrollieren*)
			IF fb_state_entry.i16_last_step <> 160 THEN
				fbFindFiles.eCmd := 0;
			(*Dateien im Verzeichnis durchzählen*)
			ELSE
				fbFindFiles.eCmd := 1;
			END_IF
			fbFindFiles.bExecute := TRUE;
		END_IF

		(*-----------------------Weiterschaltbedingungen----------------------------*)
		IF fbFindFiles.bBusy THEN
			fb_state_entry.i16_next_step:=160;
		END_IF

		IF fb_state_entry.X THEN
			fbFindFiles.bExecute := FALSE;
		END_IF

(*=======================================================*)
	160:(*Prüfe, ob Maschinen Datei vorhanden ist*)
		(*-----------------------Weiterschaltbedingungen----------------------------*)
		(*letzte Datei im Verzeichnis erreicht*)
		IF fbFindFiles.bEOE AND NOT fbFindFiles.bBusy AND NOT fbFindFiles.bError  THEN
			IF fbFindFiles.nFindFiles <> 0 OR b_datei_vorhanden  THEN
				(*Datei vorhanden -> muss eingelesen werden*)
				fb_state_entry.i16_next_step:=170;
			ELSE
				(*Datei noch nicht vorhanden -> kann nicht eingelesen werden*)
				fb_state_entry.i16_next_step:=999;
			END_IF
		(*Datei wurde im Verzeichnis gefunden*)
		ELSIF NOT fbFindFiles.bBusy AND NOT fbFindFiles.bError  THEN
			IF fbFindFiles.nFindFiles <> 0  THEN
				(*Datei vorhanden -> muss eingelesen werden*)
				b_datei_vorhanden := TRUE;
				fb_state_entry.i16_next_step := 150;
			END_IF
		ELSIF fbFindFiles.bError THEN
			nErrId := fbFindFiles.nErrID;
			sm_fehler_lesen_wartungsprotokoll := TRUE;
			fb_state_entry.i16_next_step:=FEHLER;
		END_IF

		IF fb_state_entry.X THEN
			b_lesen_komplett := FALSE;
		END_IF

(*=======================================================*)
	170:	(* Lesen Maschinen Wartungsprotokoll *)
		IF fb_state_entry.E THEN
			b_datei_vorhanden := FALSE;
			sPathName := CONCAT(s_wartung_path_md,sFileName_md);
			fb_xml_srv_read.sSymName := '.gst_datensatz.st_wartungsprotokoll.st_wartung_md';
			fb_xml_srv_read.sXPath := '/root/gst_datensatz.st_wartungsprotokoll.st_wartung_md';
			fb_xml_srv_read.bExecute:= TRUE;
		END_IF

		(*-----------------------Weiterschaltbedingungen----------------------------*)
		IF fb_xml_srv_read.bBusy THEN
			fb_state_entry.i16_next_step := 180;
		END_IF

		IF fb_state_entry.X THEN
			fb_xml_srv_read.bExecute:= FALSE;
		END_IF

(*=======================================================*)
	180:
		(*-----------------------Weiterschaltbedingungen----------------------------*)
		(*Lesen erfolgreich*)
		IF NOT fb_xml_srv_read.bError AND NOT fb_xml_srv_read.bBusy THEN
			fb_state_entry.i16_next_step := 999;
		ELSIF fb_xml_srv_read.bError THEN
			nErrId:=fb_xml_srv_read.nErrId;
			sm_fehler_lesen_Wartungsprotokoll:=TRUE;
			fb_state_entry.i16_next_step := FEHLER;
		END_IF

(*=======================================================*)
	200:(*Schreibe Werkzeug Wartungsdatei*)
		IF fb_state_entry.E THEN
			sPathName := CONCAT(s_wartung_path_wkz,sFileName_wkz);
			sPathName:=CONCAT(sPathName,'.xml');
			fb_xml_srv_write.sSymName := '.gst_datensatz.st_wartungsprotokoll.st_wartung_wkz';
			fb_xml_srv_write.sXPath := '/root/gst_datensatz.st_wartungsprotokoll.st_wartung_wkz';
			fb_xml_srv_write.bExecute:= TRUE;
		END_IF

		(*-----------------------Weiterschaltbedingungen----------------------------*)
		IF fb_xml_srv_write.bBusy THEN
			fb_state_entry.i16_next_step := 210;
		END_IF

		IF fb_state_entry.X THEN
			fb_xml_srv_write.bExecute:= FALSE;
		END_IF

(*=======================================================*)
	210:
		(*-----------------------Weiterschaltbedingungen----------------------------*)
		IF NOT fb_xml_srv_write.bError AND NOT fb_xml_srv_write.bBusy THEN
			st_wartungsprotokoll_wkz_copy.st_wartung_wkz:= gst_datensatz.st_wartungsprotokoll.st_wartung_wkz ;
			fb_state_entry.i16_next_step := 999;
		END_IF


		IF fb_xml_srv_write.bError  THEN
			nErrId:=fb_xml_srv_write.nErrId;
			sm_fehler_schreiben_Wartungsprotokoll:=TRUE;
			fb_state_entry.i16_next_step := FEHLER;
		END_IF


(*===================Schrittkette====================================*)
	250:(*Schreibe Maschinen Wartungsdatei*)
		IF fb_state_entry.E THEN
			sPathName := CONCAT(s_wartung_path_md,sFileName_md);
			fb_xml_srv_write.sSymName := '.gst_datensatz.st_wartungsprotokoll.st_wartung_md';
			fb_xml_srv_write.sXPath := '/root/gst_datensatz.st_wartungsprotokoll.st_wartung_md';
			fb_xml_srv_write.bExecute:= TRUE;
		END_IF

		(*-----------------------Weiterschaltbedingungen----------------------------*)
		IF fb_xml_srv_write.bBusy THEN
			fb_state_entry.i16_next_step := 260;
		END_IF

		IF fb_state_entry.X THEN
			fb_xml_srv_write.bExecute:= FALSE;
		END_IF

(*=======================================================*)
	260:
		(*-----------------------Weiterschaltbedingungen----------------------------*)
		IF NOT fb_xml_srv_write.bError AND NOT fb_xml_srv_write.bBusy THEN
			st_wartungsprotokoll_md_copy.st_wartung_md:= gst_datensatz.st_wartungsprotokoll.st_wartung_md ;
			fb_state_entry.i16_next_step := 999;
		END_IF

		IF fb_xml_srv_write.bError  THEN
			nErrId:=fb_xml_srv_write.nErrId;
			sm_fehler_schreiben_Wartungsprotokoll:=TRUE;
			fb_state_entry.i16_next_step := FEHLER;
		END_IF

(*=======================================================*)
	300:(*Speichern der Wartungsdateien auf den Server*)
		IF 	fb_state_entry.E THEN
			fb_nt_start_process.START:=TRUE;
		END_IF

		IF fb_nt_start_process.BUSY THEN
			fb_state_entry.i16_next_step := 310;
			fb_nt_start_process.START:=FALSE;
		END_IF

(*=======================================================*)
	310:
		(*-----------------------Weiterschaltbedingungen----------------------------*)
		IF NOT fb_nt_start_process.ERR AND NOT fb_nt_start_process.BUSY THEN
			fb_state_entry.i16_next_step := 999;
		END_IF

		IF fb_nt_start_process.ERR THEN
			nErrId:=fb_nt_start_process.ERRID;
			sm_fehler_speichern_Wartungsprotokoll;
			fb_state_entry.i16_next_step:=FEHLER;
		END_IF

(*=======================================================*)
	400:(*Prüfe, ob Werkzeug Datei vorhanden ist*)
		IF fb_state_entry.E THEN
			sPathName := CONCAT(s_wartung_path_wkz,sFileName_wkz);
			sPathName:=CONCAT(sPathName,'_RESET');
			sPathName:=CONCAT(sPathName,'.xml');
			(*Erste Datei im Verzeichnis kontrollieren*)
			IF fb_state_entry.i16_last_step <> 410 THEN
				fbFindFiles.eCmd := 0;
			(*Dateien im Verzeichnis durchzählen*)
			ELSE
				fbFindFiles.eCmd := 1;
			END_IF
			fbFindFiles.bExecute := TRUE;
		END_IF

		(*-----------------------Weiterschaltbedingungen----------------------------*)
		IF fbFindFiles.bBusy THEN
			fb_state_entry.i16_next_step:=410;
		END_IF

		IF fb_state_entry.X THEN
			fbFindFiles.bExecute := FALSE;
		END_IF

(*=======================================================*)
	410:(*Prüfe, ob Werkzeug Datei vorhanden ist*)
		(*-----------------------Weiterschaltbedingungen----------------------------*)
		(*letzte Datei im Verzeichnis erreicht*)
		IF fbFindFiles.bEOE AND NOT fbFindFiles.bBusy AND NOT fbFindFiles.bError  THEN
			IF fbFindFiles.nFindFiles <> 0 OR b_datei_vorhanden  THEN
				(*Datei vorhanden -> darf nicht neu geschrieben werden*)
				fb_state_entry.i16_next_step:=999;
			ELSE
				(*Datei noch nicht vorhanden -> muss erstellt werden*)
				fb_state_entry.i16_next_step := 420;
			END_IF
		(*Datei wurde im Verzeichnis gefunden*)
		ELSIF NOT fbFindFiles.bBusy AND NOT fbFindFiles.bError  THEN
			IF fbFindFiles.nFindFiles <> 0  THEN
				(*Datei vorhanden -> muss eingelesen werden*)
				b_datei_vorhanden := TRUE;
				fb_state_entry.i16_next_step := 400;
			END_IF
		ELSIF fbFindFiles.bError THEN
			nErrId := fbFindFiles.nErrID;
			sm_fehler_lesen_Wartungsprotokoll := TRUE;
			fb_state_entry.i16_next_step:=FEHLER;
		END_IF

(*=======================================================*)
	420:(*Schreibe Werkzeug Reset Wartungsdatei*)
		IF fb_state_entry.E THEN
			sPathName := CONCAT(s_wartung_path_wkz,sFileName_wkz);
			sPathName:=CONCAT(sPathName,'_RESET');
			sPathName:=CONCAT(sPathName,'.xml');
			fb_xml_srv_write.sSymName := '.gst_datensatz.st_wartungsprotokoll.st_wartung_wkz';
			fb_xml_srv_write.sXPath := '/root/gst_datensatz.st_wartungsprotokoll.st_wartung_wkz';
			fb_xml_srv_write.bExecute:= TRUE;
		END_IF

		(*-----------------------Weiterschaltbedingungen----------------------------*)
		IF fb_xml_srv_write.bBusy THEN
			fb_state_entry.i16_next_step := 430;
		END_IF

		IF fb_state_entry.X THEN
			fb_xml_srv_write.bExecute:= FALSE;
		END_IF

(*=======================================================*)
	430:
		(*-----------------------Weiterschaltbedingungen----------------------------*)
		IF NOT fb_xml_srv_write.bError AND NOT fb_xml_srv_write.bBusy THEN
			i32_bestueckhubzaehler_md_copy:=gst_datensatz.st_md.i32_bestueckhubzaehler;
			s_aktuelles_wkz_copy:=gst_datensatz.st_md.s_aktuelles_wkz;
			gst_datensatz.st_wartungsprotokoll.st_wartung_wkz.hubzaehler := 0;
			i32_bestueckhubzaehler_wkz_copy := 0;
			fb_state_entry.i16_next_step := 999;
		END_IF

		IF fb_xml_srv_write.bError  THEN
			nErrId:=fb_xml_srv_write.nErrId;
			sm_fehler_schreiben_Wartungsprotokoll:=TRUE;
			fb_state_entry.i16_next_step := FEHLER;
		END_IF


(*=======================================================*)
	999:	(* Ende - Befehl wurde korrekt abgearbeitet *)
		IF fb_state_entry.E THEN
			b_datei_vorhanden := FALSE;
			st_ctrl_out.b_busy := FALSE;
			st_ctrl_out.b_fertig := TRUE;
			i16_auftrag := KEIN_WARTUNG_AUFTRAG;
			fb_state_entry.i16_next_step := BEREIT;
		END_IF

(*=======================================================*)
	FEHLER: (* Fehler *)
		IF fb_state_entry.E THEN
			i16_auftrag := KEIN_WARTUNG_AUFTRAG;
			st_ctrl_out.b_bereit := FALSE;
			st_ctrl_out.b_busy := FALSE;
			st_ctrl_out.b_fertig := FALSE;
			st_ctrl_out.b_fehler := TRUE;
			fb_ton_quitt.IN := FALSE;
		END_IF

		(*-----------------------Weiterschaltbedingungen----------------------------*)
		IF st_ctrl_in.b_quitt AND NOT fb_state_entry.E THEN
			st_ctrl_out.b_fehler := FALSE;
			fb_ton_quitt.IN := TRUE;
		END_IF

		IF fb_ton_quitt.Q THEN
			fb_ton_quitt.IN := FALSE;
			fb_state_entry.i16_next_step := INIT;
		END_IF
END_CASE

fb_state_entry(i16_pos:= 2 );

(* ======================================Subkomponenten======================================== *)

IF st_config.b_config_fertig THEN
	garr_stoermeldungen[st_config.i16_meld_startindex + 0] := sm_fehler_schreiben_Wartungsprotokoll;
	garr_stoermeldungen[st_config.i16_meld_startindex + 1] := sm_fehler_lesen_Wartungsprotokoll;
	garr_stoermeldungen[st_config.i16_meld_startindex + 2] := sm_fehler_speichern_Wartungsprotokoll;
	garr_stoermeldungen[st_config.i16_meld_startindex + 3] := FALSE;
	garr_stoermeldungen[st_config.i16_meld_startindex + 4] := FALSE;
	garr_stoermeldungen[st_config.i16_meld_startindex + 5] := FALSE;
	garr_stoermeldungen[st_config.i16_meld_startindex + 6] := FALSE;
	garr_stoermeldungen[st_config.i16_meld_startindex + 7] := FALSE;
	garr_stoermeldungen[st_config.i16_meld_startindex + 8] := FALSE;
	garr_stoermeldungen[st_config.i16_meld_startindex + 9] := FALSE;
	garr_stoermeldungen[st_config.i16_meld_startindex + 10] := FALSE;
	garr_stoermeldungen[st_config.i16_meld_startindex + 11] := FALSE;
	garr_stoermeldungen[st_config.i16_meld_startindex + 12] := FALSE;
	garr_stoermeldungen[st_config.i16_meld_startindex + 13] := FALSE;
	garr_stoermeldungen[st_config.i16_meld_startindex + 14] := FALSE;
	garr_stoermeldungen[st_config.i16_meld_startindex + 15] := FALSE;
	garr_stoermeldungen[st_config.i16_meld_startindex + 16] := FALSE;
	garr_stoermeldungen[st_config.i16_meld_startindex + 17] := FALSE;
	garr_stoermeldungen[st_config.i16_meld_startindex + 18] := FALSE;
	garr_stoermeldungen[st_config.i16_meld_startindex + 19] := FALSE;

	garr_betriebsmeldungen[st_config.i16_meld_startindex + 0] :=FALSE;
	garr_betriebsmeldungen[st_config.i16_meld_startindex + 1] := FALSE;
	garr_betriebsmeldungen[st_config.i16_meld_startindex + 2] := FALSE;
	garr_betriebsmeldungen[st_config.i16_meld_startindex + 3] := FALSE;
	garr_betriebsmeldungen[st_config.i16_meld_startindex + 4] := FALSE;
	garr_betriebsmeldungen[st_config.i16_meld_startindex + 5] := FALSE;
	garr_betriebsmeldungen[st_config.i16_meld_startindex + 6] := FALSE;
	garr_betriebsmeldungen[st_config.i16_meld_startindex + 7] := FALSE;
	garr_betriebsmeldungen[st_config.i16_meld_startindex + 8] := FALSE;
	garr_betriebsmeldungen[st_config.i16_meld_startindex + 9] := FALSE;
	garr_betriebsmeldungen[st_config.i16_meld_startindex + 10] := FALSE;
	garr_betriebsmeldungen[st_config.i16_meld_startindex + 11] := FALSE;
	garr_betriebsmeldungen[st_config.i16_meld_startindex + 12] := FALSE;
	garr_betriebsmeldungen[st_config.i16_meld_startindex + 13] := FALSE;
	garr_betriebsmeldungen[st_config.i16_meld_startindex + 14] := FALSE;
	garr_betriebsmeldungen[st_config.i16_meld_startindex + 15] := FALSE;
	garr_betriebsmeldungen[st_config.i16_meld_startindex + 16] := FALSE;
	garr_betriebsmeldungen[st_config.i16_meld_startindex + 17] := FALSE;
	garr_betriebsmeldungen[st_config.i16_meld_startindex + 18] := FALSE;
	garr_betriebsmeldungen[st_config.i16_meld_startindex + 19] := FALSE;
END_IF
END_PROGRAM
ACTION auto_speichern_laden:
(*========================================================================================*)
(*ohne Timer wurde nicht immer gespeichert*)
fb_ton_end(
	IN:=  i16_auftrag = KEIN_WARTUNG_AUFTRAG,
	PT:= t#100ms,
	Q=> ,
	ET=> );


(*Werkzeug Daten speichern*)
IF	fb_ton_end.Q AND gi16_maschinenstatusinfo <> STATUS_MASCHINE_ARBEITET AND
	(MEMCMP(ADR(st_wartungsprotokoll_wkz_copy.st_wartung_wkz), ADR(gst_datensatz.st_wartungsprotokoll.st_wartung_wkz), SIZEOF(st_wartungsprotokoll_wkz_copy.st_wartung_wkz)) <> 0 ) THEN
	i16_auftrag:=SCHREIBE_WARTUNGSPROTOKOLL_WKZ;
END_IF


(*Maschinen Daten speichern*)
IF	fb_ton_end.Q AND gi16_maschinenstatusinfo <> STATUS_MASCHINE_ARBEITET AND
	(MEMCMP(ADR(st_wartungsprotokoll_md_copy.st_wartung_md), ADR(gst_datensatz.st_wartungsprotokoll.st_wartung_md), SIZEOF(st_wartungsprotokoll_md_copy.st_wartung_md)) <> 0 ) THEN
	i16_auftrag:=SCHREIBE_WARTUNGSPROTOKOLL_MD;
END_IF

(*Button in der Oberfläche für das Reseten nach der Wartung*)
IF fb_ton_end.Q AND gi16_maschinenstatusinfo <> STATUS_MASCHINE_ARBEITET AND fb_r_trig_reset_wkz.Q THEN
	i16_auftrag:=SCHREIBE_WARTUNGSPROTOKOLL_WKZ_RESET;
END_IF
END_ACTION
ACTION fb_Aufrufe:
fb_xml_srv_read(
	sNetId:= ,
	ePath:= PATH_GENERIC,
	nMode:= XMLSRV_SKIPMISSING,
	sFilePath:=sPathName,
	bExecute:= ,
	tTimeout:= t#20s,
	bBusy=> ,
	bError=> ,
	nErrId=> );


fb_xml_srv_write(
	sNetId:= '',
	ePath:= PATH_GENERIC,
	nMode:= XMLSRV_ADDMISSING,
	sFilePath:=sPathName,
	bExecute:= ,
	tTimeout:= t#10s,
	bBusy=> ,
	bError=> ,
	nErrId=> );


fbFindFiles(
	bExecute	:= ,
	sNetId		:= '',
	sPathName	:= sPathName,
	pFindList		:= ADR(file),
	cbFindList	:= SIZEOF(file),
	tTimeout	:= t#1s );


fb_nt_start_process(
	NETID:= '',
	PATHSTR:= 'C:\Windows\System32\wscript.exe',
	DIRNAME:=s_tools_path,
	COMNDLINE:=CONCAT(visu.s_akt_sprache,'_Wartung_nach_server.vbs'),	 	(*CONCAT(visu.s_akt_sprache,'_Wartung_nach_server.vbs'),		'de_Wartung_nach_server.vbs', 	*)
	START:= ,
	TMOUT:= DEFAULT_ADS_TIMEOUT,
	BUSY=> ,
	ERR=> ,
	ERRID=> nErrId);



FB_GetHostName(
	sNetID:= '127.0.0.1.1.1',
	bExecute:= , 
	tTimeout:= , 
	bBusy=> ,
	bError=> ,
	nErrID=> , 
	sHostName=> );
END_ACTION
ACTION FileName_erstellen:
(*Name für Werkzeug Datei*)
sFileName_wkz:='';
sFileName_wkz:=CONCAT(sFileName_wkz,gst_datensatz.st_md.s_aktuelles_wkz);
sFileName_wkz:=CONCAT(sFileName_wkz,s_Trennstelle);
sFileName_wkz:=CONCAT(sFileName_wkz,FB_GetHostName.sHostName);
sFileName_wkz:=CONCAT(sFileName_wkz,s_Trennstelle);
sFileName_wkz:=CONCAT(sFileName_wkz,gstr_datum);

(*Name für Maschinen Datei*)
sFileName_md:='';
sFileName_md:=CONCAT(sFileName_md,FB_GetHostName.sHostName);
sFileName_md:=CONCAT(sFileName_md,'.xml');
END_ACTION
ACTION Zaehler:
IF fb_state_entry.i16_step = BEREIT THEN
	(*Übergabe der aktuellen Betriebsstunden der Zelle in die Wartungsstruktur*)
	gst_datensatz.st_wartungsprotokoll.st_wartung_md.betriebsstunden := gst_datensatz.st_md.i32_betriebssekundenzaehler/ 3600;

	(*Übergabe des aktuellen Hubzählers der Zelle in die Wartungsstruktur*)
	gst_datensatz.st_wartungsprotokoll.st_wartung_md.hubzaehler := gst_datensatz.st_md.i32_bestueckhubzaehler;

	(*Übergabe der aktuell produzierten Stecker der Zelle in die Wartungsstruktur*)
	gst_datensatz.st_wartungsprotokoll.st_wartung_md.produzierte_stecker := gst_datensatz.st_md.produzierte_Stecker;

	(*Übergabe des aktuellen Hubzählers des benutzten Werkzeugs an die Wartungsstruktur*)
	gst_datensatz.st_wartungsprotokoll.st_wartung_wkz.hubzaehler := i32_bestueckhubzaehler_wkz_copy + (gst_datensatz.st_md.i32_bestueckhubzaehler-i32_bestueckhubzaehler_md_copy);
END_IF
END_ACTION

(* POU MAINs/MAIN_FAST, ST *)
PROGRAM MAIN_FAST
VAR
END_VAR
CASE gst_datensatz.st_md.i16_typ_zelle OF
	KEINE_ZELLE:
		ST_Safetyprogramm(
			st_config:= safety.st_config,
			st_ctrl_in:= safety.st_ctrl.in,
			st_visu:= safety.st_visu,
			st_ctrl_out=> safety.st_ctrl.out);

		ST_Betriebsfreigaben(
			st_config:= betriebsfreigaben.st_config,
			st_ctrl_in:= betriebsfreigaben.st_ctrl.in,
			b_lampe_stoerung:= ,
			b_lampe_produktion:= ,
			e_steuerung_ein:= ST_Safetyprogramm.se_steuerung_ein,
			st_ctrl_out=> betriebsfreigaben.st_ctrl.out);

		nockenschaltwerk_bestueckachse.fb(
			r_achsposition:= virtuelle_master_achse.NcToPlc.ModuloActPos,
			r_achsgeschwindigkeit:= virtuelle_master_achse.NcToPlc.ActVelo * 60 / 360,
			i16_verfahrrichtung_achse_extern:=  ,
			b_verfahrrichtungsauswertung_extern:= FALSE,
			i16_art_der_achse:= RUND,
			st_config:= nockenschaltwerk_bestueckachse.st_config,
			arr_nocken:= gst_datensatz.st_wkz.nockenschaltwerk_bestueckachse.arr_nocken,
			st_visu:= visu);

	BESTUECKZELLE_1700:
		ST_Safetyprogramm(
			st_config:= safety.st_config,
			st_ctrl_in:= safety.st_ctrl.in,
			st_visu:= safety.st_visu,
			st_ctrl_out=> safety.st_ctrl.out);

		ST_Betriebsfreigaben(
			st_config:= betriebsfreigaben.st_config,
			st_ctrl_in:= betriebsfreigaben.st_ctrl.in,
			b_lampe_stoerung:= ,
			b_lampe_produktion:= ,
			e_steuerung_ein:= ST_Safetyprogramm.se_steuerung_ein,
			st_ctrl_out=> betriebsfreigaben.st_ctrl.out);

		nockenschaltwerk_bestueckachse.fb(
			r_achsposition:= virtuelle_master_achse.NcToPlc.ModuloActPos,
			r_achsgeschwindigkeit:= virtuelle_master_achse.NcToPlc.ActVelo * 60 / 360,
			i16_verfahrrichtung_achse_extern:=  ,
			b_verfahrrichtungsauswertung_extern:= FALSE,
			i16_art_der_achse:= RUND,
			st_config:= nockenschaltwerk_bestueckachse.st_config,
			arr_nocken:= gst_datensatz.st_wkz.nockenschaltwerk_bestueckachse.arr_nocken,
			st_visu:= visu);

		ST_Virtuelle_Masterachse(
			st_config_achse:= axis_virt_master.st_config,
			e_ls_bandende_re := ST_Bandwechsel_Kontroller.e_ls_bandende_re,
			e_ls_bandende_li	:= ST_Bandwechsel_Kontroller.e_ls_bandende_li,
			st_ctrl_in:= axis_virt_master.st_ctrl.in,
			e_steuerung_ein:= ST_Safetyprogramm.se_steuerung_ein,
			e_ba_mit_bedingungen:= ST_Safetyprogramm.se_ba_mit_bedingungen,
			st_visu:= axis_virt_master.st_visu,
			st_visu_virtuell:= axis_virt_master.st_visu,
			st_ctrl_out=> axis_virt_master.st_ctrl.out,
			b_materialmangel=> ST_LampeMaterialMangel.b_materialmangel[2],
			b_materialmangel2=> ST_LampeMaterialMangel.b_materialmangel[6]);

		CASE gst_datensatz.st_wkz.i16_typ_bandeinzug OF
			KEIN_EINZUG:
				;
			STANDARD_2FACH_V2:
				;
			BANDWECHSLER_V2:
				;
			SERVO:
				ST_Servobandeinzug(
					st_config_achse:= axis_bandeinzug_achse.st_config,
					st_ctrl_in:= axis_bandeinzug_achse.st_ctrl.in,
					e_steuerung_ein:= ST_Safetyprogramm.se_steuerung_ein,
					e_ba_mit_bedingungen:= ST_Safetyprogramm.se_ba_mit_bedingungen,
					e_tuere_vorne_offen:= ST_Safetyprogramm.se_tuere_vorne_offen,
					e_tuere_hinten_offen:= ST_Safetyprogramm.se_tuere_hinten_offen,
					st_visu:= axis_bandeinzug_achse.st_visu,
					st_ctrl_out=> axis_bandeinzug_achse.st_ctrl.out);
		END_CASE

		ST_WkzAbsicherung(
			st_config:= wkz_absicherung.st_config,
			st_ctrl_in:= wkz_absicherung.st_ctrl.in,
			st_visu:= wkz_absicherung.st_visu,
			st_ctrl_out=> wkz_absicherung.st_ctrl.out);

		ST_Einpress_Kontroller(
			st_config:= einpresskraft_kontroller.st_config,
			st_ctrl_in:= einpresskraft_kontroller.st_ctrl.in,
			lr_achsposition:= bestueckachse.NcToPlc.ModuloActPos,
			st_visu:= einpresskraft_kontroller.st_visu,
			st_einpressen:= gst_datensatz.st_band.st_einpressen,
			st_ctrl_out=> einpresskraft_kontroller.st_ctrl.out);


		ST_Bandeinzug_Kontroller_1700(
			st_config:= bandeinzug_kontroller.st_config,
			st_ctrl_in:= bandeinzug_kontroller.st_ctrl.in,
			st_visu:= bandeinzug_kontroller.st_visu,
			st_ctrl_out=> bandeinzug_kontroller.st_ctrl.out);

		ST_Zylinder_Fast();

	BESTUECKZELLE_1720:
		ST_Safetyprogramm(
			st_config:= safety.st_config,
			st_ctrl_in:= safety.st_ctrl.in,
			st_visu:= safety.st_visu,
			st_ctrl_out=> safety.st_ctrl.out);

		ST_Betriebsfreigaben(
			st_config:= betriebsfreigaben.st_config,
			st_ctrl_in:= betriebsfreigaben.st_ctrl.in,
			b_lampe_stoerung:= ,
			b_lampe_produktion:= ,
			e_steuerung_ein:= ST_Safetyprogramm.se_steuerung_ein,
			st_ctrl_out=> betriebsfreigaben.st_ctrl.out);
		
		nockenschaltwerk_bestueckachse.fb(
			r_achsposition:= virtuelle_master_achse.NcToPlc.ModuloActPos,
			r_achsgeschwindigkeit:= virtuelle_master_achse.NcToPlc.ActVelo * 60 / 360,
			i16_verfahrrichtung_achse_extern:=  ,
			b_verfahrrichtungsauswertung_extern:= FALSE,
			i16_art_der_achse:= RUND,
			st_config:= nockenschaltwerk_bestueckachse.st_config,
			arr_nocken:= gst_datensatz.st_wkz.nockenschaltwerk_bestueckachse.arr_nocken,
			st_visu:= visu);

		ST_Virtuelle_Masterachse(
			st_config_achse:= axis_virt_master.st_config,
			e_ls_bandende_re := ST_Bandeinzug_Kontroller_1720.e_ls_bandende_re,
			e_ls_bandende_li	:= ST_Bandeinzug_Kontroller_1720.e_ls_bandende_li,
			st_ctrl_in:= axis_virt_master.st_ctrl.in,
			e_steuerung_ein:= ST_Safetyprogramm.se_steuerung_ein,
			e_ba_mit_bedingungen:= ST_Safetyprogramm.se_ba_mit_bedingungen,
			st_visu:= axis_virt_master.st_visu,
			st_visu_virtuell:= axis_virt_master.st_visu,
			st_ctrl_out=> axis_virt_master.st_ctrl.out,
			b_materialmangel=> ST_LampeMaterialMangel.b_materialmangel[2],
			b_materialmangel2=> ST_LampeMaterialMangel.b_materialmangel[6]);

		ST_WkzAbsicherung(
			st_config:= wkz_absicherung.st_config,
			st_ctrl_in:= wkz_absicherung.st_ctrl.in,
			st_visu:= wkz_absicherung.st_visu,
			st_ctrl_out=> wkz_absicherung.st_ctrl.out);

		ST_Bandeinzug_Kontroller_1720(
			st_config:= bandeinzug_kontroller.st_config,
			st_ctrl_in:= bandeinzug_kontroller.st_ctrl.in,
			st_visu:= bandeinzug_kontroller.st_visu,
			st_ctrl_out=> bandeinzug_kontroller.st_ctrl.out);

		ST_Zylinder_Fast();

	RASTERFOLIE:
		ST_Safetyprogramm(
			st_config:= safety.st_config,
			st_ctrl_in:= safety.st_ctrl.in,
			st_visu:= safety.st_visu,
			st_ctrl_out=> safety.st_ctrl.out);
	
		ST_Betriebsfreigaben(
			st_config:= betriebsfreigaben.st_config,
			st_ctrl_in:= betriebsfreigaben.st_ctrl.in,
			b_lampe_stoerung:= ,
			b_lampe_produktion:= ,
			e_steuerung_ein:= ST_Safetyprogramm.se_steuerung_ein,
			st_ctrl_out=> betriebsfreigaben.st_ctrl.out);
		
		nockenschaltwerk_bestueckachse.fb(
			r_achsposition:= virtuelle_master_achse.NcToPlc.ModuloActPos,
			r_achsgeschwindigkeit:= virtuelle_master_achse.NcToPlc.ActVelo * 60 / 360,
			i16_verfahrrichtung_achse_extern:=  ,
			b_verfahrrichtungsauswertung_extern:= FALSE,
			i16_art_der_achse:= RUND,
			st_config:= nockenschaltwerk_bestueckachse.st_config,
			arr_nocken:= gst_datensatz.st_wkz.nockenschaltwerk_bestueckachse.arr_nocken,
			st_visu:= visu);

		ST_Virtuelle_Masterachse(
			st_config_achse:= axis_virt_master.st_config,
			e_ls_bandende_re := ST_Bandwechsel_Kontroller.e_ls_bandende_re,
			e_ls_bandende_li	:= ST_Bandwechsel_Kontroller.e_ls_bandende_li,
			st_ctrl_in:= axis_virt_master.st_ctrl.in,
			e_steuerung_ein:= ST_Safetyprogramm.se_steuerung_ein,
			e_ba_mit_bedingungen:= ST_Safetyprogramm.se_ba_mit_bedingungen,
			st_visu:= axis_virt_master.st_visu,
			st_visu_virtuell:= axis_virt_master.st_visu,
			st_ctrl_out=> axis_virt_master.st_ctrl.out,
			b_materialmangel=> ST_LampeMaterialMangel.b_materialmangel[2],
			b_materialmangel2=> ST_LampeMaterialMangel.b_materialmangel[6]);
END_CASE
END_PROGRAM

(* POU Gemeinsamkeiten17xx/Betriebsfreigaben/ST_Betriebsfreigaben, ST *)
PROGRAM ST_Betriebsfreigaben
VAR_INPUT
	st_config							: struct_config;
	st_ctrl_in							: struct_ctrl_in;
	b_lampe_stoerung				: BOOL;
	b_lampe_produktion				: BOOL;
	e_steuerung_ein					: BOOL;
END_VAR
VAR_OUTPUT
	st_ctrl_out						: struct_ctrl_out;
END_VAR
VAR
	fb_tof_druck						: TOF;
	fb_tof_druck_hublift_links			: TOF;
	fb_ton_ls_schalter_ausgeloest		: TON;
	fb_ton_temperatur_schaltschrank	: TON;
	fb_ton_ueberstrom_haspe			: TON;
	fb_ton_quitt						: TON;
	fb_ton_wz						: TON;
	fb_state_entry						: ST_StateEntry;
	sm_druckwaechter  				: BOOL := FALSE;
	sm_druckwaechter_hublift_links		: BOOL := FALSE;
	sm_schaltschrank 					: BOOL := FALSE;
	sm_ls_schalter 					: BOOL := FALSE;
	sm_haube_offen 					: BOOL := FALSE;
	sm_ueberstrom_haspel			: BOOL := FALSE;

	bm_schaltschrank 					: BOOL := FALSE;

	e_temperatur_schaltschrank 		AT %I* : BOOL;
	e_ls_schalter_ausgeloest 			AT %I* : BOOL;

	e_ueberstrom_haspel				AT %I* : BOOL;
	a_lampe_steuerung 				AT %Q* : BOOL;
	e_druckwaechter					AT %I* : BOOL;
	e_druckwaechter_hublift_links		AT %I* : BOOL;
	a_lampe_stoerung 				AT %Q* : BOOL;
	a_lampe_produktion 				AT %Q* : BOOL;
END_VAR
fb_tof_druck(IN:=e_druckwaechter , PT:= t#500ms, Q=> , ET=> );
fb_tof_druck_hublift_links(IN:=e_druckwaechter_hublift_links , PT:= t#500ms, Q=> , ET=> );
fb_ton_ls_schalter_ausgeloest(IN:=NOT e_ls_schalter_ausgeloest  , PT:= t#200ms, Q=> , ET=> );
fb_ton_temperatur_schaltschrank(IN:=NOT e_temperatur_schaltschrank  , PT:= t#200ms, Q=> , ET=> );
fb_ton_ueberstrom_haspe(IN:=NOT e_ueberstrom_haspel , PT:= t#200ms, Q=> , ET=> );

fb_ton_wz(IN:= , PT:= t#500ms, Q=> , ET=> );
fb_ton_quitt(IN:= , PT:= t#50ms, Q=> , ET=> );

a_lampe_steuerung := e_steuerung_ein ;
a_lampe_stoerung := b_lampe_stoerung;
a_lampe_produktion := b_lampe_produktion;

bm_schaltschrank:=fb_ton_temperatur_schaltschrank.Q;
ST_LampeMaterialMangel.b_materialmangel[4]:=bm_schaltschrank;

(*=======================Schrittkette=======================*)
fb_state_entry(
	i16_next_step:= ,
	i16_pos:= 1,
	s_debugtext:= ,
	E=> ,
	X=> ,
	i16_step=> ,
	i16_last_step=> );

CASE fb_state_entry.i16_step OF
(*=======================================================*)
	INIT_OBJ:
		IF st_config.b_config_fertig THEN
			fb_state_entry.i16_next_step := INIT;
		END_IF

(*=======================================================*)
	INIT:
		st_ctrl_out.b_fehler := FALSE;
		st_ctrl_out.b_bereit := FALSE;
		fb_ton_wz.IN := FALSE;
		fb_ton_quitt.IN := FALSE;
		sm_druckwaechter  := FALSE;
		sm_druckwaechter_hublift_links := FALSE;
		sm_schaltschrank  := FALSE;
		sm_ls_schalter  := FALSE;
		sm_haube_offen := FALSE;
		sm_ueberstrom_haspel := FALSE;
		bm_schaltschrank  := FALSE;
		(*-----------------------Weiterschaltbedingungen----------------------------*)
		fb_state_entry.i16_next_step := BEREIT;

(*=======================================================*)
	BEREIT:
		IF fb_state_entry.E THEN
			st_ctrl_out.b_bereit := TRUE;
		END_IF

		(*-----------------------Weiterschaltbedingungen----------------------------*)
		IF 	NOT fb_tof_druck.Q THEN
			sm_druckwaechter := TRUE;
			fb_state_entry.i16_next_step := FEHLER;
		END_IF
		IF	 fb_ton_ls_schalter_ausgeloest.Q THEN
			sm_ls_schalter := TRUE;
			fb_state_entry.i16_next_step := FEHLER;
		END_IF
		(*IF 	fb_ton_ueberstrom_foerderbaender.Q THEN
			sm_ueberstrom_foerderbaender := TRUE;
			fb_state_entry.i16_next_step := FEHLER;
		END_IF*)
		IF 	fb_ton_ueberstrom_haspe.Q THEN
			sm_ueberstrom_haspel := TRUE;
			fb_state_entry.i16_next_step := FEHLER;
		END_IF
		IF gst_datensatz.st_md.b_hublift_links_aktiv THEN
			IF NOT fb_tof_druck_hublift_links.Q THEN
				sm_druckwaechter_hublift_links := TRUE;
				fb_state_entry.i16_next_step := FEHLER;
			END_IF
		END_IF

(*		IF 	fb_ton_temperatur_schaltschrank.Q THEN
			sm_schaltschrank := TRUE;
			fb_state_entry.i16_next_step := FEHLER;
		END_IF*)

(*=======================================================*)
	FEHLER:
		IF fb_state_entry.E THEN
			st_ctrl_out.b_fehler := TRUE;
			fb_ton_quitt.IN := FALSE;
		END_IF

